// TwinCAT 3 PLC project OC_TwinCAT_EtherCAT
// Title: OC_EtherCAT
// Company: Open Commissioning
// Author: SpiraTec AG
// ProjectVersion: 1.1.8
// Description: Open Commissioning TwinCAT EtherCAT Library
// ProgramVersion: 3.1.4026.19
// libraries:
//   OC_Core, * (Open Commissioning)
//   OC_TwinSAFE, * (Open Commissioning)
//   Tc2_Math, * (Beckhoff Automation GmbH)
//   Tc2_Standard, * (Beckhoff Automation GmbH)
//   Tc2_System, * (Beckhoff Automation GmbH)
//   Tc3_Module, * (Beckhoff Automation GmbH)
//   TcUnit, * (www.tcunit.org)
// project tree:
//   Devices/Drives/DS402/ E_DS402_State.TcDUT, FB_DS402_CSP.TcPOU, FB_DS402_FSM.TcPOU, ST_DS402_CSP_Config.TcDUT, ST_DS402_ControlWord.TcDUT, ST_DS402_CSP_Status.TcDUT, ST_DS402_CSP_Control.TcDUT, ST_DS402_StatusWord.TcDUT
//   Devices/Drives/Mitsubishi/ FB_Mitsubishi_MRJ4TM.TcPOU, ST_Mitsubishi_MRJ4TM_Config.TcDUT, ST_Mitsubishi_MRJ4TM_Control.TcDUT, ST_Mitsubishi_MRJ4TM_Status.TcDUT
//   Devices/Drives/Sercos/ E_Sercos_State.TcDUT, FB_Sercos_FSM.TcPOU, FB_Sercos_VC.TcPOU, ST_Sercos_VC.TcDUT, ST_Sercos_VC_Config.TcDUT, ST_Sercos_VC_Control.TcDUT, ST_Sercos_VC_Status.TcDUT, ST_Sercos_StatusWord.TcDUT, ST_Sercos_ControlWord.TcDUT
//   Devices/Terminals/ FB_Beckhoff_EK1914.TcPOU, FB_Beckhoff_EL5152.TcPOU, FB_Beckhoff_EJ1918.TcPOU, FB_Beckhoff_EL1904.TcPOU, FB_Beckhoff_EL1918.TcPOU, FB_Beckhoff_EL2904.TcPOU, FB_FSOE_19.TcPOU, ST_Baumer_Encoder.TcDUT, ST_Beckhoff_16DI.TcDUT, ST_Beckhoff_16DO.TcDUT (not stored), ST_Beckhoff_2AI.TcDUT (not stored), ST_Beckhoff_4AI.TcDUT (not stored), ST_Beckhoff_4AO.TcDUT, ST_Beckhoff_4DI_4DO.TcDUT (not stored), ST_Beckhoff_8DI.TcDUT, ST_Beckhoff_4DI.TcDUT, ST_Beckhoff_8DI_8DO.TcDUT (not stored), ST_Beckhoff_8DO.TcDUT (not stored), ST_Beckhoff_4DO.TcDUT, ST_Beckhoff_EL3403.TcDUT (not stored), ST_Beckhoff_EL5002.TcDUT (not stored), ST_Beckhoff_EL9110.TcDUT (not stored), ST_Beckhoff_EL9410.TcDUT (not stored), ST_CoE402.TcDUT (not stored), ST_Gefran_GFX4.TcDUT (not stored), ST_Mitsubishi_MRJ4TM.TcDUT, ST_SEW_SimMovitrac.TcDUT (not stored)
//   Devices/Terminals/FB_Beckhoff_EL6001/ E_Beckhoff_EL6001_State.TcDUT, FB_Beckhoff_EL6001.TcPOU
//   / PlcTask.TcTTO
//   Tests/Drives/ FB_Sercos_VC_Test.TcPOU, FB_DS402_FSM_Test.TcPOU, FB_DS402_CSP_Test.TcPOU, FB_Sercos_FSM_Test.TcPOU
//   Tests/Terminals/ FB_Beckhoff_EL5152_Test.TcPOU, FB_Beckhoff_EL6001_Test.TcPOU
//   Tests/ PRG_TEST.TcPOU

CONFIGURATION OC_TwinCAT_EtherCAT
    RESOURCE PLC ON TwinCAT3
        TASK PlcTask(INTERVAL := T#1ms, PRIORITY := 30);
        PROGRAM PRG_TEST WITH PlcTask : PRG_TEST;
    END_RESOURCE
END_CONFIGURATION

// ---- Devices/Drives/DS402/E_DS402_State.TcDUT
{attribute 'qualified_only'}
{attribute 'strict'}
{attribute 'conditionalshow'}
TYPE E_DS402_State :
(
	S0_NotReadyToSwitchOn,
	S1_SwitchOnDisabled,
	S2_ReadyToSwitchOn,
	S3_SwitchedOn,
	S4_OperationEnabled,
	S5_Fault,
	S6_FaultReactionActive,
	S7_QuickStopActive
);
END_TYPE

// ---- Devices/Drives/DS402/ST_DS402_CSP_Config.TcDUT
{attribute 'pack_mode' := '0'}
TYPE ST_DS402_CSP_Config :
STRUCT	
	bForceMode			: BOOL; //Ignore process data from fieldbus.	
	bSwapProcessData	: BOOL; //Reverse process data byte order from/to fieldbus.
	fPositionOffset		: LREAL := 0.0;	
	bSyncOpMode			: BOOL := TRUE;
END_STRUCT
END_TYPE

// ---- Devices/Drives/DS402/ST_DS402_ControlWord.TcDUT
(*
	Object 6040h: Control word (DS402)	
*)
{attribute 'pack_mode' := '0'}
TYPE ST_DS402_ControlWord :
STRUCT
	b0_SwitchOn 					: BIT;
	b1_EnableVoltage				: BIT;
	b2_QuickStop					: BIT;
	b3_EnableOperation				: BIT;
	b4_OperationModeSpecific		: BIT;
	b5_OperationModeSpecific		: BIT;
	b6_OperationModeSpecific		: BIT;
	b7_FaultReset					: BIT;
	b8_Reserved						: BIT;
	b9_Reserved						: BIT;
	b10_Reserved					: BIT;
	b11_Reserved					: BIT;
	b12_Reserved					: BIT;
	b13_Reserved					: BIT;
	b14_Reserved					: BIT;
	b15_Reserved					: BIT;
END_STRUCT
END_TYPE

// ---- Devices/Drives/DS402/ST_DS402_CSP_Status.TcDUT
(*
	Status struct for Cyclic synchronous position mode(CSP)
	0x1A00 (DS402 Statusword)
	0x1A01 (DS402 Position actual value)
	0x1A04 (DS402 Following error actual value)
*)
{attribute 'pack_mode' := '0'}
TYPE ST_DS402_CSP_Status :
STRUCT
	nStatusWord 		: ST_DS402_StatusWord; //0x1A00 (DS402 Statusword)
	nActualPosition		: DINT;	//0x1A01 (DS402 Position actual value) [INC]
	nErrorPosition		: DINT;	//0x1A04 (DS402 Following error actual value) [INC]	
END_STRUCT
END_TYPE

// ---- Devices/Drives/DS402/ST_DS402_CSP_Control.TcDUT
(*
	Control struct for Cyclic synchronous position mode(CSP)
	0x1600 (DS402 Controlword)
	0x1606 (DS402 Target position)
*)
{attribute 'pack_mode' := '0'}
TYPE ST_DS402_CSP_Control :
STRUCT
	nControlWord 		: ST_DS402_ControlWord; //0x1600 (DS402 Controlword)
	nTargetPosition		: DINT;	//DS402 Target position [INC]	
END_STRUCT
END_TYPE

// ---- Devices/Drives/DS402/ST_DS402_StatusWord.TcDUT
(*
	Object 6041h: Status word (DS402)
*)
{attribute 'pack_mode' := '0'}
TYPE ST_DS402_StatusWord :
STRUCT
	b0_ReadyToSwitchOn 				: BIT; 
	b1_SwitchedOn 					: BIT; 
	b2_OperationEnabled 			: BIT; 
	b3_Fault						: BIT; 
	b4_VoltageEnabled				: BIT; 
	b5_QuickStop					: BIT;
	b6_SwitchOnDisabled				: BIT; 
	b7_Warning						: BIT; 
	b8_Synchranisation				: BIT; 
	b9_Remote						: BIT;
	b10_TargetReached				: BIT;
	b11_InternalLimitActive			: BIT; 
	b12_OperationModeSpecific		: BIT; 
	b13_OperationModeSpecific		: BIT; 
	b14_OperationModeSpecific		: BIT; 
	b15_ClosedLoopActive			: BIT;
END_STRUCT
END_TYPE

// ---- Devices/Drives/Mitsubishi/ST_Mitsubishi_MRJ4TM_Config.TcDUT
{attribute 'pack_mode' := '0'}
TYPE ST_Mitsubishi_MRJ4TM_Config :
STRUCT	
	bForceMode			: BOOL; //Ignore process data from fieldbus.	
	bSwapProcessData	: BOOL; //Reverse process data byte order from/to fieldbus.
	fPositionOffset		: LREAL := 0.0;	
	bSyncOpMode			: BOOL := TRUE;
END_STRUCT
END_TYPE

// ---- Devices/Drives/Mitsubishi/ST_Mitsubishi_MRJ4TM_Control.TcDUT
(*
	
*)
{attribute 'pack_mode' := '0'}
TYPE ST_Mitsubishi_MRJ4TM_Control :
STRUCT
	nModesOfOperation 				: SINT;
	nControlWord 					: ST_DS402_ControlWord; //0x1600 (DS402 Controlword)
	nControlID1						: UINT;
	nControlID2						: UINT;
	nControlID3						: UINT;
	nTargetPosit					: DINT;
	nTargetVeloc					: DINT;
	nVelocityLimitValue				: UDINT;
	nTargetTorque					: INT;
	nPositiveTorqueLimitValue		: UINT;
	nNegativeTorqueLimitValue 		: UINT;
	nTouchProbeFunction				: UINT;
END_STRUCT
END_TYPE

// ---- Devices/Drives/Mitsubishi/ST_Mitsubishi_MRJ4TM_Status.TcDUT
(*
	
*)
{attribute 'pack_mode' := '0'}
TYPE ST_Mitsubishi_MRJ4TM_Status :
STRUCT
	nModesOfOperationDisplay 		: SINT;
	nStatusWord 					: ST_DS402_StatusWord; //0x1A00 (DS402 Statusword)
	nStatusDO1						: UINT;
	nStatusDO2						: UINT;
	nStatusDO3						: UINT;
	nPositionActualValue			: DINT;
	nVelocityActualValue			: DINT;
	nFollowingErrorActualValue		: DINT;
	nTorqueActualValue				: INT;
	nTouchProbeStatus				: UINT;
	nTouchProbePos1PosValue			: DINT;
	nTouchProbePos1NegValue			: DINT;
	nTouchProbePos2PosValue			: DINT;
	nTouchProbePos2NegValue			: DINT;
END_STRUCT
END_TYPE

// ---- Devices/Drives/Sercos/E_Sercos_State.TcDUT
{attribute 'qualified_only'}
{attribute 'strict'}
{attribute 'conditionalshow'}
TYPE E_Sercos_State :
(
	S1_NotReadyToSwitchOn,
	S2_SwitchOnDisabled,
	S3_ReadyToSwitchOn,
	S4_SwitchOn,
	S5a_DriveInOperation,
	S5b_Halt,
	S6_QuickStop,
	S7_FaultReactionActive,
	S8_Fault
);
END_TYPE

// ---- Devices/Drives/Sercos/ST_Sercos_VC.TcDUT
{attribute 'pack_mode' := '1'} 
TYPE ST_Sercos_VC :
STRUCT
	stControl		AT %I* : ST_Sercos_VC_Control;
	stStatus		AT %Q* : ST_Sercos_VC_Status;
END_STRUCT
END_TYPE

// ---- Devices/Drives/Sercos/ST_Sercos_VC_Config.TcDUT
{attribute 'pack_mode' := '0'}
TYPE ST_Sercos_VC_Config :
STRUCT	
	bForceMode				: BOOL; //Ignore process data from fieldbus.	
	bSwapProcessData		: BOOL; //Reverse process data byte order from/to fieldbus.	
	bIsLinkOutputVelocity	: BOOL; //If TRUE, link output is velocity value
	fReferenceVelocity 		: REAL := 1000.0;
	fNormalizationFactor	: REAL := 80000;
END_STRUCT
END_TYPE

// ---- Devices/Drives/Sercos/ST_Sercos_VC_Control.TcDUT
(*
	Sercos Velocity Control
	MDT: S-0-0134 Master control word
	MDT: S-0-0036 Velocity command value
*)
{attribute 'pack_mode' := '0'}
TYPE ST_Sercos_VC_Control :
STRUCT
	nControlWord 			: ST_Sercos_ControlWord; //S-0-0134 Master control word
	nVelocityCommand		: DINT;	//S-0-0036 Velocity command value
END_STRUCT
END_TYPE

// ---- Devices/Drives/Sercos/ST_Sercos_VC_Status.TcDUT
(*
	Sercos Velocity Control
	AT: S-0-0135 Drive Status word
	AT: S-0-0051 Position feedback 1 value
*)
{attribute 'pack_mode' := '0'}
TYPE ST_Sercos_VC_Status :
STRUCT
	nStatusWord 			: ST_Sercos_StatusWord; //S-0-0135 Drive Status word
	nPositionFeedback		: DINT;	//S-0-0051 Position feedback 1 value
END_STRUCT
END_TYPE

// ---- Devices/Drives/Sercos/ST_Sercos_StatusWord.TcDUT
(*
	S-0-0135 Drive Status
	https://product-help.schneider-electric.com/Machine%20Expert/V1.2/en/ATV340SUG/ATV340SUG/STI_Software_Setup/STI_Software_Setup-22.htm#XREF_D_SE_0083227_1
*)
{attribute 'pack_mode' := '1'}
TYPE ST_Sercos_StatusWord :
STRUCT
	b0_Reserved 					: BIT;
	b1_Reserved						: BIT;
	b2_Reserved						: BIT;
	b3_CommandProcessing			: BIT; //Status command value processing if 0 = ignored
	b4_Halt							: BIT; //Drive halt, 0 = inactive, 1 = active
	b5_PositionFeedback				: BIT; //Position feedback value status (S-0-0403)
	b6_Reserved						: BIT;
	b7_QuickStop					: BIT; //Quick stop, 0 = inactive, 1 = active
	b8_Reserved						: BIT; //Reserved (=0)
	b9_Reserved						: BIT; //Reserved (=0)
	b10_OperationMode				: BIT; //0 = Primary operation mode
	b11_Reserved					: BIT;
	b12_Warning						: BIT; //Warning, 0 = No warning, 1 = Warning
	b13_Error						: BIT; //Drive shut-down error, 0 = No error, 1 = Error
	b14_ReadyToOperate				: BIT; //00 = Not ready to switch on, 01 = Switch on disabled, main power disabled
	b15_ReadyToOperate				: BIT; //10 = Switch on, 11 = Drive enabled
END_STRUCT
END_TYPE

// ---- Devices/Drives/Sercos/ST_Sercos_ControlWord.TcDUT
(*
	S-0-0134 Drive Control
	https://product-help.schneider-electric.com/Machine%20Expert/V1.2/en/ATV340SUG/ATV340SUG/STI_Software_Setup/STI_Software_Setup-21.htm#XREF_D_SE_0083221_1
*)
{attribute 'pack_mode' := '1'}
TYPE ST_Sercos_ControlWord :
STRUCT
	b0_Reserved 					: BIT;
	b1_Reserved						: BIT;
	b2_Reserved						: BIT;
	b3_Reserved						: BIT;
	b4_Reserved						: BIT;
	b5_Reserved						: BIT;
	b6_Reserved						: BIT;
	b7_Reserved						: BIT;
	b8_Reserved						: BIT; //Reserved (=0)
	b9_Reserved						: BIT; //Reserved (=0)
	b10_OperationMode				: BIT; //0 = Primary operation mode
	b11_Reserved					: BIT;
	b12_Reserved					: BIT; 
	b13_Halt						: BIT; //Drive halt, 1 --> 0 = halt, 0 --> 1 = restart
	b14_Start						: BIT; //Drive start, 1 --> 0 = Stop, 0 -> 1 = Start 
	b15_Enable						: BIT; //Drive enable, 1 --> 0 = drive disabled, 0 -> 1 = drive enabled
END_STRUCT
END_TYPE

// ---- Devices/Terminals/FB_Beckhoff_EL6001/E_Beckhoff_EL6001_State.TcDUT
{attribute 'qualified_only'}
{attribute 'strict'}
TYPE E_Beckhoff_EL6001_State :
(
	INIT,
	READY,
	TRANSMIT, 
	RECEIVE
);
END_TYPE

// ---- Devices/Terminals/ST_Baumer_Encoder.TcDUT
{attribute 'pack_mode' := '1'}
TYPE ST_Baumer_Encoder :
STRUCT
	nPosition		AT %Q*	:	UDINT;
	nWarnings		AT %Q*	:	UINT;
	nSystemTime		AT %Q*	:	UDINT; 
END_STRUCT
END_TYPE

// ---- Devices/Terminals/ST_Beckhoff_16DI.TcDUT
{attribute 'pack_mode' := '1'} 
TYPE ST_Beckhoff_16DI :
STRUCT
	bIn1	AT %Q* : BIT;
	bIn2	AT %Q* : BIT;
	bIn3	AT %Q* : BIT;
	bIn4	AT %Q* : BIT;
	bIn5	AT %Q* : BIT;
	bIn6	AT %Q* : BIT;
	bIn7	AT %Q* : BIT;
	bIn8	AT %Q* : BIT;
	bIn9	AT %Q* : BIT;
	bIn10	AT %Q* : BIT;
	bIn11	AT %Q* : BIT;
	bIn12	AT %Q* : BIT;
	bIn13	AT %Q* : BIT;
	bIn14	AT %Q* : BIT;
	bIn15	AT %Q* : BIT;
	bIn16	AT %Q* : BIT;
END_STRUCT
END_TYPE

// ---- Devices/Terminals/ST_Beckhoff_4AO.TcDUT
{attribute 'pack_mode' := '1'} 
TYPE ST_Beckhoff_4AO :
STRUCT
	nAnalogOut1	AT %I* : UINT;
	nAnalogOut2	AT %I* : UINT;
	nAnalogOut3	AT %I* : UINT;
	nAnalogOut4	AT %I* : UINT;
END_STRUCT
END_TYPE

// ---- Devices/Terminals/ST_Beckhoff_8DI.TcDUT
{attribute 'pack_mode' := '1'} 
TYPE ST_Beckhoff_8DI :
STRUCT
	bIn1	AT %Q* : BIT;
	bIn2	AT %Q* : BIT;
	bIn3	AT %Q* : BIT;
	bIn4	AT %Q* : BIT;
	bIn5	AT %Q* : BIT;
	bIn6	AT %Q* : BIT;
	bIn7	AT %Q* : BIT;
	bIn8	AT %Q* : BIT;
END_STRUCT
END_TYPE

// ---- Devices/Terminals/ST_Beckhoff_4DI.TcDUT
{attribute 'pack_mode' := '1'} 
TYPE ST_Beckhoff_4DI :
STRUCT
	bIn1	AT %Q* : BIT;
	bIn2	AT %Q* : BIT;
	bIn3	AT %Q* : BIT;
	bIn4	AT %Q* : BIT;	
END_STRUCT
END_TYPE

// ---- Devices/Terminals/ST_Beckhoff_4DO.TcDUT
{attribute 'pack_mode' := '1'} 
TYPE ST_Beckhoff_4DO :
STRUCT
	bOut1	AT %I* : BIT;
	bOut2	AT %I* : BIT;
	bOut3	AT %I* : BIT;
	bOut4	AT %I* : BIT;	
END_STRUCT
END_TYPE

// ---- Devices/Terminals/ST_Mitsubishi_MRJ4TM.TcDUT
{attribute 'pack_mode' := '1'} 
TYPE ST_Mitsubishi_MRJ4TM :
STRUCT
	nModesOfOperation 				AT %I* : SINT;
	nControlWord					AT %I* : UINT;
	nControlID1						AT %I* : UINT;
	nControlID2						AT %I* : UINT;
	nControlID3						AT %I* : UINT;
	nTargetPosit					AT %I* : DINT;
	nTargetVeloc					AT %I* : DINT;
	nVelocityLimitValue				AT %I* : UDINT;
	nTargetTorque					AT %I* : INT;
	nPositiveTorqueLimitValue		AT %I* : UINT;
	nNegativeTorqueLimitValue 		AT %I* : UINT;
	nTouchProbeFunction				AT %I* : UINT;
	
	nModesOfOperationDisplay 		AT %Q* : SINT;
	nStatusWord						AT %Q* : UINT;
	nStatusDO1						AT %Q* : UINT;
	nStatusDO2						AT %Q* : UINT;
	nStatusDO3						AT %Q* : UINT;
	nPositionActualValue			AT %Q* : DINT;
	nVelocityActualValue			AT %Q* : DINT;
	nFollowingErrorActualValue		AT %Q* : DINT;
	nTorqueActualValue				AT %Q* : INT;
	nTouchProbeStatus				AT %Q* : UINT;
	nTouchProbePos1PosValue			AT %Q* : DINT;
	nTouchProbePos1NegValue			AT %Q* : DINT;
	nTouchProbePos2PosValue			AT %Q* : DINT;
	nTouchProbePos2NegValue			AT %Q* : DINT;
END_STRUCT
END_TYPE

// ---- Tests/PRG_TEST.TcPOU
PROGRAM PRG_TEST
VAR	
	FB_System	: FB_System;
	FB_Beckhoff_EL5152_Test : FB_Beckhoff_EL5152_Test;
	FB_Beckhoff_EL6001_Test : FB_Beckhoff_EL6001_Test;
	FB_DS402_FSM_Test : FB_DS402_FSM_Test;	
	FB_DS402_CSP_Test : FB_DS402_CSP_Test; 
	FB_Sercos_FSM_Test : FB_Sercos_FSM_Test;
	FB_Sercos_VC_Test : FB_Sercos_VC_Test;
END_VAR

FB_System();
TcUnit.RUN();

END_PROGRAM

// ---- Tests/Terminals/FB_Beckhoff_EL5152_Test.TcPOU
FUNCTION_BLOCK FB_Beckhoff_EL5152_Test EXTENDS TcUnit.FB_TestSuite
VAR
	_fbDevice 	: FB_Beckhoff_EL5152;
	_nExpected 	: UINT;
	_nResult 	: UINT;
END_VAR

TEST('nCounter1');
_nExpected := 111;
_fbDevice.nValue1 := _nExpected;
_fbDevice();
_nResult := _fbDevice.Counter1;
AssertEquals(Expected := _nExpected,
             Actual := _nResult,
             Message := 'nCounter1 value is not correct');	
TEST_FINISHED();

TEST('nCounter2');
_nExpected := 112;
_fbDevice.nValue2 := _nExpected;
_fbDevice();
_nResult := _fbDevice.Counter2;
AssertEquals(Expected := _nExpected,
             Actual := _nResult,
             Message := 'nCounter2 value is not correct');	
TEST_FINISHED();


TEST('nStatus1');
_nExpected := 4;
_fbDevice.Control1 := _nExpected;
_fbDevice();
_nResult := _fbDevice.Status1;
AssertEquals(Expected := _nExpected,
             Actual := _nResult,
             Message := 'nStatus1 value is not correct');	
TEST_FINISHED();

TEST('nStatus2');
_nExpected := 4;
_fbDevice.Control2 := _nExpected;
_fbDevice();
_nResult := _fbDevice.Status2;
AssertEquals(Expected := _nExpected,
             Actual := _nResult,
             Message := 'nStatus2 value is not correct');	
TEST_FINISHED();

END_FUNCTION_BLOCK

// ---- Devices/Terminals/FB_Beckhoff_EL5152.TcPOU
FUNCTION_BLOCK FB_Beckhoff_EL5152
VAR_INPUT
	nValue1		: UINT;
	nValue2		: UINT;
END_VAR
VAR
	nControl1		AT %I* : UINT;
	nSetCounter1	AT %I* : UINT;
	nControl2		AT %I* : UINT;
	nSetCounter2	AT %I* : UINT;
	
	nStatus1		AT %Q* : UINT;
	nCounter1		AT %Q* : UINT;	
	nPeriod1    	AT %Q* : UDINT;
	nStatus2		AT %Q* : UINT;
	nCounter2		AT %Q* : UINT;
	nPeriod2    	AT %Q* : UDINT;
END_VAR

nStatus1.2 := nControl1.2;
nStatus2.2 := nControl2.2;

nCounter1 := nValue1;
nCounter2 := nValue2;

PROPERTY INTERNAL Control1 : UINT
SET
nControl1 := Control1;
END_SET
END_PROPERTY

PROPERTY INTERNAL Control2 : UINT
SET
nControl2 := Control2;
END_SET
END_PROPERTY

PROPERTY INTERNAL Counter1 : UINT
GET
Counter1 := nCounter1;
END_GET
END_PROPERTY

PROPERTY INTERNAL Counter2 : UINT
GET
Counter2 := nCounter2;
END_GET
END_PROPERTY

PROPERTY INTERNAL Period1 : UDINT
GET
Period1 := nPeriod1;
END_GET
END_PROPERTY

PROPERTY INTERNAL Period2 : UDINT
GET
Period2 := nPeriod2;
END_GET
END_PROPERTY

PROPERTY INTERNAL SetCounter1 : UINT
SET
nSetCounter1 := SetCounter1;
END_SET
END_PROPERTY

PROPERTY INTERNAL SetCounter2 : UINT
SET
nSetCounter2 := SetCounter2;
END_SET
END_PROPERTY

PROPERTY INTERNAL Status1 : UINT
GET
Status1 := nStatus1;
END_GET
END_PROPERTY

PROPERTY INTERNAL Status2 : UINT
GET
Status2 := nStatus2;
END_GET
END_PROPERTY

END_FUNCTION_BLOCK

// ---- Tests/Terminals/FB_Beckhoff_EL6001_Test.TcPOU
FUNCTION_BLOCK FB_Beckhoff_EL6001_Test EXTENDS TcUnit.FB_TestSuite
VAR
	_fbDevice 	: FB_Beckhoff_EL6001;
	_nExpected 	: UINT;
	_nResult 	: UINT;
END_VAR

TestProperties();
TestState();

METHOD TestProperties : REFERENCE TO FB_Test
VAR
	bExpected 		: BOOL;
	bResult 		: BOOL;
END_VAR
TEST('TransmitRequest FALSE');
bExpected := FALSE; 
_fbDevice();
_fbDevice.Control := 0;
_fbDevice();
bResult := _fbDevice.TransmitRequest;
AssertEquals(Expected := bExpected,
             Actual := bResult,
             Message := 'TransmitRequest value is not correct');		
TEST_FINISHED();

TEST('TransmitRequest TRUE');
bExpected := TRUE; 
_fbDevice();
_fbDevice.Control := 1;
_fbDevice();
bResult := _fbDevice.TransmitRequest;
AssertEquals(Expected := bExpected,
             Actual := bResult,
             Message := 'TransmitRequest value is not correct');		
TEST_FINISHED();

TEST('ReceiveAccepted FALSE');
bExpected := FALSE; 
_fbDevice();
_fbDevice.Control := 0;
_fbDevice();
bResult := _fbDevice.ReceiveAccepted;
AssertEquals(Expected := bExpected,
             Actual := bResult,
             Message := 'ReceiveAccepted value is not correct');		
TEST_FINISHED();

TEST('ReceiveAccepted TRUE');
bExpected := TRUE; 
_fbDevice();
_fbDevice.Control := 2;
_fbDevice();
bResult := _fbDevice.ReceiveAccepted;
AssertEquals(Expected := bExpected,
             Actual := bResult,
             Message := 'ReceiveAccepted value is not correct');		
TEST_FINISHED();

TEST('InitRequest TRUE');
bExpected := TRUE; 
_fbDevice();
_fbDevice.Control := 4;
_fbDevice();
bResult := _fbDevice.InitRequest;
AssertEquals(Expected := bExpected,
             Actual := bResult,
             Message := 'InitRequest value is not correct');		
TEST_FINISHED();

TEST('SendContinuous TRUE');
bExpected := TRUE; 
_fbDevice.Control := 0;
_fbDevice();
_fbDevice.Control := 9;
_fbDevice();
bResult := _fbDevice.SendContinuous;
AssertEquals(Expected := bExpected,
             Actual := bResult,
             Message := 'SendContinuous value is not correct');		
TEST_FINISHED();
END_METHOD

METHOD TestState : REFERENCE TO FB_Test
VAR
	bResult 		: BOOL;
	nDataSend 		:  ARRAY[0..50] OF BYTE;
END_VAR
TEST('Transition: INIT - READY');
_fbDevice.Control := 0;
_fbDevice.State := E_Beckhoff_EL6001_State.INIT;	
_fbDevice();

AssertTRUE(_fbDevice.State = E_Beckhoff_EL6001_State.READY, 'State value is not correct');
	
TEST_FINISHED();

TEST('Transition: READY - TRANSMIT');
_fbDevice.Control := 0;
_fbDevice.State := E_Beckhoff_EL6001_State.READY;	
_fbDevice();

_fbDevice.Control := 257;
_fbDevice();

AssertTRUE(_fbDevice.State = E_Beckhoff_EL6001_State.TRANSMIT, 'State value is not correct');
	
TEST_FINISHED();

TEST('Transition: READY - RECEIVE');
_fbDevice.Control := 0;
_fbDevice.State := E_Beckhoff_EL6001_State.READY;	
_fbDevice();

_fbDevice.bSend := TRUE;
_fbDevice.pDataIn := ADR(nDataSend);
_fbDevice.nLength := 1;
_fbDevice.Control := 1;
_fbDevice();

_fbDevice.bSend := FALSE;
_fbDevice.nLength := 0;

AssertTRUE(_fbDevice.State = E_Beckhoff_EL6001_State.RECEIVE, 'State value is not correct');
TEST_FINISHED();
END_METHOD

END_FUNCTION_BLOCK

// ---- Devices/Terminals/FB_Beckhoff_EL6001/FB_Beckhoff_EL6001.TcPOU
FUNCTION_BLOCK FB_Beckhoff_EL6001
VAR_INPUT
	bSend				: BOOL;
	nLength				: UINT;
	pDataIn				: POINTER TO BYTE; //Data to send
	pDataOut			: POINTER TO BYTE; //Received data when nDataAvailable > 0.
END_VAR

VAR_OUTPUT
	bBusy				: BOOL;
	nDataAvailable		: INT; //Received bytes. Only available for one cycle.
END_VAR

VAR
	nControl			AT %I* : UINT;
	nDataOut			AT %I* : ARRAY[0..21] OF USINT;
	nStatus				AT %Q* : UINT;
	nDataIn				AT %Q* : ARRAY[0..21] OF USINT;
END_VAR

VAR
	_nControlByte			: BYTE;
	_nOutLength				: BYTE;	
	_bTransmitRequest		: BOOL;
	_bReceiveAccecpted		: BOOL;
	_bInitRequest			: BOOL;
	_bSendContinuous		: BOOL;
	
	_bTransmitAccepted		: BOOL;
	_bReceiveRequest		: BOOL;
	_bInitAccepted			: BOOL;
	_bBufferFull			: BOOL;
	_bParityError			: BOOL;
	_bFramingError			: BOOL;
	_bOverrunError			: BOOL;
	_nInLength				: BYTE;
	
	_nPendingLength			: UINT;
	_nOffsetNext			: UINT;
	
	_eState					: E_Beckhoff_EL6001_State;
	_trigSend				: R_TRIG;
END_VAR

(* Receive control word *)
	_bTransmitRequest 	:= nControl.0 <> _nControlByte.0;
	_bReceiveAccecpted 	:= nControl.1 <> _nControlByte.1;
	_bInitRequest		:= nControl = 4;
	_bSendContinuous		:= nControl.3 AND NOT _nControlByte.0;	
	_nControlByte 		:= F_GetLByte(nControl);
	_nOutLength 			:= F_GetHByte(nControl);

(* Initialize *)
	IF _bInitRequest THEN
		_eState := E_Beckhoff_EL6001_State.INIT;			
	END_IF
	
CASE _eState OF
	E_Beckhoff_EL6001_State.INIT:
		_bTransmitAccepted 	:= FALSE;
		_bReceiveRequest		:= FALSE;
		_bInitAccepted		:= TRUE;
		_bBufferFull			:= FALSE;
		_bParityError		:= FALSE;
		_bFramingError		:= FALSE;
		_bOverrunError		:= FALSE;
		_nInLength			:= 0;
		nDataAvailable		:= 0;
		
		// -> INIT_READY
		IF nControl = 0 THEN
			_bInitAccepted := FALSE;		
			_eState := E_Beckhoff_EL6001_State.READY;
		END_IF

	E_Beckhoff_EL6001_State.READY:
		nDataAvailable := 0;

		// -> TRANSMIT
		IF _bTransmitRequest AND _nOutLength > 0 AND _nOutLength < 23 THEN
			_eState := E_Beckhoff_EL6001_State.TRANSMIT;
			RETURN;
		END_IF
		
		_trigSend(CLK := bSend);
		
		// -> RECEIVE
		IF _trigSend.Q AND nLength > 0 AND pDataIn <> 0 THEN
			_bReceiveRequest := NOT _bReceiveRequest;
			_nPendingLength := nLength;
			_nInLength := UINT_TO_BYTE(MIN(22, _nPendingLength));
			memcpy(ADR(nDataIn), pDataIn, _nInLength);		
			_eState := E_Beckhoff_EL6001_State.RECEIVE;
		END_IF	
		
	E_Beckhoff_EL6001_State.TRANSMIT:
		IF pDataOut <> 0 THEN
			memcpy(pDataOut, ADR(nDataOut), _nOutLength);
		END_IF
		_bTransmitAccepted := NOT _bTransmitAccepted;
		nDataAvailable := _nOutLength;
		_eState := E_Beckhoff_EL6001_State.READY;
		
	E_Beckhoff_EL6001_State.RECEIVE:
		IF _bReceiveAccecpted THEN
			_nOffsetNext := _nInLength;
			_nPendingLength := _nPendingLength - _nOffsetNext;
			IF _nPendingLength = 0 THEN
				_eState := E_Beckhoff_EL6001_State.READY;
			END_IF
			IF _nPendingLength > 0 THEN
				_bReceiveRequest := NOT _bReceiveRequest;
				_nInLength := UINT_TO_BYTE(MIN(22, _nPendingLength));
				memcpy(ADR(nDataIn), pDataIn + _nOffsetNext, _nInLength);
				_eState := E_Beckhoff_EL6001_State.RECEIVE;
			END_IF				
		END_IF
	
END_CASE

bBusy := _eState <> E_Beckhoff_EL6001_State.READY;
	
(* Send status word *)
	nStatus.0			:= _bTransmitAccepted;
	nStatus.1			:= _bReceiveRequest;
	nStatus.2			:= _bInitAccepted;
	nStatus.3			:= _bBufferFull;
	nStatus.4			:= _bParityError;
	nStatus.5			:= _bFramingError;
	nStatus.6			:= _bOverrunError;
	memcpy(ADR(nStatus) + 1, ADR(_nInLength), 1);

PROPERTY INTERNAL BufferFull : BOOl
GET
BufferFull := _bBufferFull;
END_GET
END_PROPERTY

PROPERTY INTERNAL Control : UINT
SET
nControl := Control;
END_SET
END_PROPERTY

PROPERTY INTERNAL FramingError : BOOl
GET
FramingError := _bFramingError;
END_GET
END_PROPERTY

PROPERTY INTERNAL InitAccepted : BOOl
GET
InitAccepted := _bInitAccepted;
END_GET
END_PROPERTY

PROPERTY INTERNAL InitRequest : BOOl
GET
InitRequest := _bInitRequest;
END_GET
END_PROPERTY

PROPERTY INTERNAL OverrunError : BOOl
GET
OverrunError := _bOverrunError;
END_GET
END_PROPERTY

PROPERTY INTERNAL ParityError : BOOl
GET
ParityError := _bParityError;
END_GET
END_PROPERTY

PROPERTY INTERNAL ReceiveAccepted : BOOl
GET
ReceiveAccepted := _bReceiveAccecpted;
END_GET
END_PROPERTY

PROPERTY INTERNAL ReceiveRequest : BOOl
GET
ReceiveRequest := _bReceiveRequest;
END_GET
END_PROPERTY

PROPERTY INTERNAL SendContinuous : BOOl
GET
SendContinuous := _bSendContinuous;
END_GET
END_PROPERTY

PROPERTY INTERNAL State : E_Beckhoff_EL6001_State
GET
State := _eState;
END_GET
SET
_eState := State;
END_SET
END_PROPERTY

PROPERTY INTERNAL TransmitAccepted : BOOl
GET
TransmitAccepted := _bTransmitAccepted;
END_GET
END_PROPERTY

PROPERTY INTERNAL TransmitRequest : BOOl
GET
TransmitRequest := _bTransmitRequest;
END_GET
END_PROPERTY

END_FUNCTION_BLOCK

// ---- Tests/Drives/FB_DS402_FSM_Test.TcPOU
FUNCTION_BLOCK FB_DS402_FSM_Test EXTENDS TcUnit.FB_TestSuite

TestStateS0();
TestStateS1();
TestStateS2();
TestStateS3();
TestStateS4();
TestStateS5();
TestStateS6();
TestStateS7();
TestEnableSequence();

METHOD PRIVATE GetDisableCommand : ST_DS402_ControlWord
GetDisableCommand.b0_SwitchOn := TRUE;
GetDisableCommand.b1_EnableVoltage := TRUE;
GetDisableCommand.b2_QuickStop := TRUE;
GetDisableCommand.b3_EnableOperation := FALSE;
GetDisableCommand.b7_FaultReset := FALSE;
END_METHOD

METHOD PRIVATE GetDisableVoltageCommand : ST_DS402_ControlWord
GetDisableVoltageCommand.b1_EnableVoltage := FALSE;
GetDisableVoltageCommand.b7_FaultReset := FALSE;
END_METHOD

METHOD PRIVATE GetEnableCommand : ST_DS402_ControlWord
GetEnableCommand.b0_SwitchOn := TRUE;
GetEnableCommand.b1_EnableVoltage := TRUE;
GetEnableCommand.b2_QuickStop := TRUE;
GetEnableCommand.b3_EnableOperation := TRUE;
GetEnableCommand.b7_FaultReset := FALSE;
END_METHOD

METHOD PRIVATE GetQuickStopCommand : ST_DS402_ControlWord
GetQuickStopCommand.b2_QuickStop := FALSE;
GetQuickStopCommand.b7_FaultReset := FALSE;
END_METHOD

METHOD PRIVATE GetShotdownCommand : ST_DS402_ControlWord
GetShotdownCommand.b0_SwitchOn := FALSE;
GetShotdownCommand.b1_EnableVoltage := TRUE;
GetShotdownCommand.b2_QuickStop := TRUE;
GetShotdownCommand.b7_FaultReset := FALSE;
END_METHOD

METHOD PRIVATE GetSwitchOnCommand : ST_DS402_ControlWord
GetSwitchOnCommand.b0_SwitchOn := TRUE;
GetSwitchOnCommand.b1_EnableVoltage := TRUE;
GetSwitchOnCommand.b2_QuickStop := TRUE;
GetSwitchOnCommand.b7_FaultReset := FALSE;
END_METHOD

METHOD TestEnableSequence : BOOL
VAR
	fbDS402 			: FB_DS402_FSM;
	stExpectedStatus 	: ST_DS402_StatusWord; 
	nMask 				: WORD;
	nResult 			: WORD;
	bResult 			: BOOL;
	nActualState		: INT;
	nExpectedState		: INT;
END_VAR
TEST('Enable S1');

fbDS402();
nExpectedState := E_DS402_State.S1_SwitchOnDisabled;
nActualState := fbDS402.eState;

AssertEquals(Expected := nExpectedState,
             Actual := nActualState,
             Message := 'State is not correct');	 
TEST_FINISHED();

TEST('Enable S2');
fbDS402.stControl.b1_EnableVoltage := TRUE;
fbDS402.stControl.b2_QuickStop := TRUE;

fbDS402();
nExpectedState := E_DS402_State.S2_ReadyToSwitchOn;
nActualState := fbDS402.eState;

AssertEquals(Expected := nExpectedState,
             Actual := nActualState,
             Message := 'State is not correct');	 
TEST_FINISHED();

TEST('Enable S3');
fbDS402.stControl.b0_SwitchOn := TRUE;

fbDS402();
nExpectedState := E_DS402_State.S3_SwitchedOn;
nActualState := fbDS402.eState;

AssertEquals(Expected := nExpectedState,
             Actual := nActualState,
             Message := 'State is not correct');	 
TEST_FINISHED();

TEST('Enable S4');
fbDS402.stControl.b3_EnableOperation := TRUE;

fbDS402();
nExpectedState := E_DS402_State.S4_OperationEnabled;
nActualState := fbDS402.eState;

AssertEquals(Expected := nExpectedState,
             Actual := nActualState,
             Message := 'State is not correct');	 
TEST_FINISHED();

TEST('Disable S4');
fbDS402.stControl.b3_EnableOperation := FALSE;

fbDS402();
nExpectedState := E_DS402_State.S3_SwitchedOn;
nActualState := fbDS402.eState;

AssertEquals(Expected := nExpectedState,
             Actual := nActualState,
             Message := 'State is not correct');	 
TEST_FINISHED();

TEST('Disable S3');
fbDS402.stControl.b0_SwitchOn := FALSE;

fbDS402();
nExpectedState := E_DS402_State.S2_ReadyToSwitchOn;
nActualState := fbDS402.eState;

AssertEquals(Expected := nExpectedState,
             Actual := nActualState,
             Message := 'State is not correct');	 
TEST_FINISHED();

TEST('Disable S2');
fbDS402.stControl.b1_EnableVoltage := FALSE;
fbDS402.stControl.b2_QuickStop := FALSE;

fbDS402();
nExpectedState := E_DS402_State.S1_SwitchOnDisabled;
nActualState := fbDS402.eState;

AssertEquals(Expected := nExpectedState,
             Actual := nActualState,
             Message := 'State is not correct');	 
TEST_FINISHED();
END_METHOD

METHOD TestStateS0 : BOOL
VAR
	fbDS402 			: FB_DS402_FSM;
	stExpectedStatus 	: ST_DS402_StatusWord; 
	nMask 				: WORD;
	nResult 			: WORD;
	bResult 			: BOOL;
	nActualState		: INT;
	nExpectedState		: INT;
END_VAR
TEST('Set State S0');
fbDS402.eState := E_DS402_State.S0_NotReadyToSwitchOn;
fbDS402();

stExpectedStatus.b0_ReadyToSwitchOn 		:= FALSE;
stExpectedStatus.b1_SwitchedOn 				:= FALSE;
stExpectedStatus.b2_OperationEnabled		:= FALSE;
stExpectedStatus.b3_Fault					:= FALSE;
stExpectedStatus.b4_VoltageEnabled			:= FALSE;
stExpectedStatus.b6_SwitchOnDisabled 		:= FALSE;

MEMCPY(ADR(nMask), ADR(stExpectedStatus), 2);
nResult := (2#01011111 AND fbDS402.nStatus);

AssertEquals(Expected := nMask,
             Actual := nResult,
             Message := 'Value is not correct');	 
TEST_FINISHED();

TEST('Transition S0>S1');
fbDS402.eState := E_DS402_State.S0_NotReadyToSwitchOn;
fbDS402();
fbDS402();

nExpectedState := E_DS402_State.S1_SwitchOnDisabled;
nActualState := fbDS402.eState;

AssertEquals(Expected := nExpectedState,
             Actual := nActualState,
             Message := 'State is not correct');	 
TEST_FINISHED();
END_METHOD

METHOD TestStateS1 : BOOL
VAR
	fbDS402 			: FB_DS402_FSM;
	stExpectedStatus 	: ST_DS402_StatusWord; 
	nMask 				: WORD;
	nResult 			: WORD;
	bResult 			: BOOL;
	nActualState		: INT;
	nExpectedState		: INT;
END_VAR
TEST('Set State S1');
fbDS402.eState := E_DS402_State.S1_SwitchOnDisabled;
fbDS402();

stExpectedStatus.b0_ReadyToSwitchOn 		:= FALSE;
stExpectedStatus.b1_SwitchedOn 				:= FALSE;
stExpectedStatus.b2_OperationEnabled		:= FALSE;
stExpectedStatus.b3_Fault					:= FALSE;
stExpectedStatus.b4_VoltageEnabled			:= FALSE;
stExpectedStatus.b6_SwitchOnDisabled 		:= TRUE;

MEMCPY(ADR(nMask), ADR(stExpectedStatus), 2);
nResult := (2#01011111 AND fbDS402.nStatus);

AssertEquals(Expected := nMask,
             Actual := nResult,
             Message := 'Value is not correct');	 
TEST_FINISHED();

TEST('Transition S1>S2');
fbDS402.eState := E_DS402_State.S1_SwitchOnDisabled;
fbDS402.stControl := GetShotdownCommand();
fbDS402();

nExpectedState := E_DS402_State.S2_ReadyToSwitchOn;
nActualState := fbDS402.eState;


AssertEquals(Expected := nExpectedState,
             Actual := nActualState,
             Message := 'State is not correct');	 
TEST_FINISHED();
END_METHOD

METHOD TestStateS2 : BOOL
VAR
	fbDS402 			: FB_DS402_FSM;
	stExpectedStatus 	: ST_DS402_StatusWord; 
	nMask 				: WORD;
	nResult 			: WORD;
	bResult 			: BOOL;
	nActualState		: INT;
	nExpectedState		: INT;
END_VAR
TEST('Set State S2');
fbDS402.eState := E_DS402_State.S2_ReadyToSwitchOn;
fbDS402();

stExpectedStatus.b0_ReadyToSwitchOn 		:= TRUE;
stExpectedStatus.b1_SwitchedOn 				:= FALSE;
stExpectedStatus.b2_OperationEnabled		:= FALSE;
stExpectedStatus.b3_Fault					:= FALSE;
stExpectedStatus.b4_VoltageEnabled			:= TRUE;
stExpectedStatus.b5_QuickStop 				:= TRUE; 
stExpectedStatus.b6_SwitchOnDisabled 		:= FALSE;

MEMCPY(ADR(nMask), ADR(stExpectedStatus), 2);
nResult := (2#01111111 AND fbDS402.nStatus);

AssertEquals(Expected := nMask,
             Actual := nResult,
             Message := 'Value is not correct');	 
TEST_FINISHED();

TEST('Transition S2>S6');
fbDS402.eState := E_DS402_State.S2_ReadyToSwitchOn;
fbDS402.bError := TRUE;
fbDS402();
fbDS402.ResetError();

nExpectedState := E_DS402_State.S6_FaultReactionActive;
nActualState := fbDS402.eState;

AssertEquals(Expected := nExpectedState,
             Actual := nActualState,
             Message := 'State is not correct');	 
TEST_FINISHED();

TEST('Transition S2>S1_1');
fbDS402.eState := E_DS402_State.S2_ReadyToSwitchOn;
fbDS402.stControl := GetDisableVoltageCommand();
fbDS402();

nExpectedState := E_DS402_State.S1_SwitchOnDisabled;
nActualState := fbDS402.eState;

AssertEquals(Expected := nExpectedState,
             Actual := nActualState,
             Message := 'State is not correct');	 
TEST_FINISHED();

TEST('Transition S2>S1_2');
fbDS402.eState := E_DS402_State.S2_ReadyToSwitchOn;
fbDS402.stControl := GetQuickStopCommand();
fbDS402.stControl.b1_EnableVoltage := TRUE;
fbDS402();

nExpectedState := E_DS402_State.S1_SwitchOnDisabled;
nActualState := fbDS402.eState;

AssertEquals(Expected := nExpectedState,
             Actual := nActualState,
             Message := 'State is not correct');	 
TEST_FINISHED();

TEST('Transition S2>S3');
fbDS402.eState := E_DS402_State.S2_ReadyToSwitchOn;
fbDS402.stControl := GetSwitchOnCommand();
fbDS402();

nExpectedState := E_DS402_State.S3_SwitchedOn;
nActualState := fbDS402.eState;

AssertEquals(Expected := nExpectedState,
             Actual := nActualState,
             Message := 'State is not correct');	 
TEST_FINISHED();
END_METHOD

METHOD TestStateS3 : BOOL
VAR
	fbDS402 			: FB_DS402_FSM;
	stExpectedStatus 	: ST_DS402_StatusWord; 
	nMask 				: WORD;
	nResult 			: WORD;
	bResult 			: BOOL;
	nActualState		: INT;
	nExpectedState		: INT;
END_VAR
TEST('Set State S3');
fbDS402.eState := E_DS402_State.S3_SwitchedOn;
fbDS402();

stExpectedStatus.b0_ReadyToSwitchOn 		:= TRUE;
stExpectedStatus.b1_SwitchedOn 				:= TRUE;
stExpectedStatus.b2_OperationEnabled		:= FALSE;
stExpectedStatus.b3_Fault					:= FALSE;
stExpectedStatus.b5_QuickStop 				:= TRUE; 
stExpectedStatus.b6_SwitchOnDisabled 		:= FALSE;

MEMCPY(ADR(nMask), ADR(stExpectedStatus), 2);
nResult := (2#01101111 AND fbDS402.nStatus);

AssertEquals(Expected := nMask,
             Actual := nResult,
             Message := 'Value is not correct');	 
TEST_FINISHED();

TEST('Transition S3>S6');
fbDS402.eState := E_DS402_State.S3_SwitchedOn;
fbDS402.bError := TRUE;
fbDS402();
fbDS402.ResetError();

nExpectedState := E_DS402_State.S6_FaultReactionActive;
nActualState := fbDS402.eState;

AssertEquals(Expected := nExpectedState,
             Actual := nActualState,
             Message := 'State is not correct');	 
TEST_FINISHED();

TEST('Transition S3>S1_1');
fbDS402.eState := E_DS402_State.S3_SwitchedOn;
fbDS402.stControl := GetDisableVoltageCommand();
fbDS402();

nExpectedState := E_DS402_State.S1_SwitchOnDisabled;
nActualState := fbDS402.eState;

AssertEquals(Expected := nExpectedState,
             Actual := nActualState,
             Message := 'State is not correct');	 
TEST_FINISHED();

TEST('Transition S3>S1_2');
fbDS402.eState := E_DS402_State.S3_SwitchedOn;
fbDS402.stControl := GetQuickStopCommand();
fbDS402.stControl.b1_EnableVoltage := TRUE;
fbDS402();

nExpectedState := E_DS402_State.S1_SwitchOnDisabled;
nActualState := fbDS402.eState;

AssertEquals(Expected := nExpectedState,
             Actual := nActualState,
             Message := 'State is not correct');	 
TEST_FINISHED();

TEST('Transition S3>S2');
fbDS402.eState := E_DS402_State.S3_SwitchedOn;
fbDS402.stControl := GetShotdownCommand();
fbDS402();

nExpectedState := E_DS402_State.S2_ReadyToSwitchOn;
nActualState := fbDS402.eState;

AssertEquals(Expected := nExpectedState,
             Actual := nActualState,
             Message := 'State is not correct');	 
TEST_FINISHED();

TEST('Transition S3>S4');
fbDS402.eState := E_DS402_State.S3_SwitchedOn;
fbDS402.stControl := GetEnableCommand();
fbDS402();

nExpectedState := E_DS402_State.S4_OperationEnabled;
nActualState := fbDS402.eState;

AssertEquals(Expected := nExpectedState,
             Actual := nActualState,
             Message := 'State is not correct');	 
TEST_FINISHED();
END_METHOD

METHOD TestStateS4 : BOOL
VAR
	fbDS402 			: FB_DS402_FSM;
	stExpectedStatus 	: ST_DS402_StatusWord; 
	nMask 				: WORD;
	nResult 			: WORD;
	bResult 			: BOOL;
	nActualState		: INT;
	nExpectedState		: INT;
END_VAR
TEST('Set State S4');
fbDS402.eState := E_DS402_State.S4_OperationEnabled;
fbDS402();

stExpectedStatus.b0_ReadyToSwitchOn 		:= TRUE;
stExpectedStatus.b1_SwitchedOn 				:= TRUE;
stExpectedStatus.b2_OperationEnabled		:= TRUE;
stExpectedStatus.b3_Fault					:= FALSE;
stExpectedStatus.b5_QuickStop 				:= TRUE; 
stExpectedStatus.b6_SwitchOnDisabled 		:= FALSE;

MEMCPY(ADR(nMask), ADR(stExpectedStatus), 2);
nResult := (2#01101111 AND fbDS402.nStatus);

AssertEquals(Expected := nMask,
             Actual := nResult,
             Message := 'Value is not correct');	 
TEST_FINISHED();

TEST('Transition S4>S6');
fbDS402.eState := E_DS402_State.S4_OperationEnabled;
fbDS402.bError := TRUE;
fbDS402();
fbDS402.ResetError();

nExpectedState := E_DS402_State.S6_FaultReactionActive;
nActualState := fbDS402.eState;

AssertEquals(Expected := nExpectedState,
             Actual := nActualState,
             Message := 'State is not correct');	 
TEST_FINISHED();

TEST('Transition S4>S1');
fbDS402.eState := E_DS402_State.S4_OperationEnabled;
fbDS402.stControl := GetDisableVoltageCommand();
fbDS402();

nExpectedState := E_DS402_State.S1_SwitchOnDisabled;
nActualState := fbDS402.eState;

AssertEquals(Expected := nExpectedState,
             Actual := nActualState,
             Message := 'State is not correct');	 
TEST_FINISHED();

TEST('Transition S4>S2');
fbDS402.eState := E_DS402_State.S4_OperationEnabled;
fbDS402.stControl := GetShotdownCommand();
fbDS402();

nExpectedState := E_DS402_State.S2_ReadyToSwitchOn;
nActualState := fbDS402.eState;

AssertEquals(Expected := nExpectedState,
             Actual := nActualState,
             Message := 'State is not correct');	 
TEST_FINISHED();

TEST('Transition S4>S3');
fbDS402.eState := E_DS402_State.S4_OperationEnabled;
fbDS402.stControl := GetDisableCommand();
fbDS402();

nExpectedState := E_DS402_State.S3_SwitchedOn;
nActualState := fbDS402.eState;

AssertEquals(Expected := nExpectedState,
             Actual := nActualState,
             Message := 'State is not correct');	 
TEST_FINISHED();

TEST('Transition S4>S7');
fbDS402.eState := E_DS402_State.S4_OperationEnabled;
fbDS402.stControl := GetQuickStopCommand();
fbDS402.stControl.b1_EnableVoltage := TRUE;
fbDS402();

nExpectedState := E_DS402_State.S7_QuickStopActive;
nActualState := fbDS402.eState;

AssertEquals(Expected := nExpectedState,
             Actual := nActualState,
             Message := 'State is not correct');	 
TEST_FINISHED();
END_METHOD

METHOD TestStateS5 : BOOL
VAR
	fbDS402 			: FB_DS402_FSM;
	stExpectedStatus 	: ST_DS402_StatusWord; 
	nMask 				: WORD;
	nResult 			: WORD;
	bResult 			: BOOL;
	nActualState		: INT;
	nExpectedState		: INT;
END_VAR
TEST('Set State S5');
fbDS402.eState := E_DS402_State.S5_Fault;
fbDS402();

stExpectedStatus.b0_ReadyToSwitchOn 		:= FALSE;
stExpectedStatus.b1_SwitchedOn 				:= FALSE;
stExpectedStatus.b2_OperationEnabled		:= FALSE;
stExpectedStatus.b3_Fault					:= TRUE;
stExpectedStatus.b6_SwitchOnDisabled 		:= FALSE;

MEMCPY(ADR(nMask), ADR(stExpectedStatus), 2);
nResult := (2#01001111 AND fbDS402.nStatus);

AssertEquals(Expected := nMask,
             Actual := nResult,
             Message := 'Value is not correct');	 
TEST_FINISHED();

TEST('Transition S5>S1');
fbDS402.eState := E_DS402_State.S5_Fault;
fbDS402.stControl.b7_FaultReset := TRUE;
fbDS402();
fbDS402.stControl.b7_FaultReset := FALSE;

nExpectedState := E_DS402_State.S1_SwitchOnDisabled;
nActualState := fbDS402.eState;

AssertEquals(Expected := nExpectedState,
             Actual := nActualState,
             Message := 'State is not correct');	 
TEST_FINISHED();
END_METHOD

METHOD TestStateS6 : BOOL
VAR
	fbDS402 			: FB_DS402_FSM;
	stExpectedStatus 	: ST_DS402_StatusWord; 
	nMask 				: WORD;
	nResult 			: WORD;
	bResult 			: BOOL;
	nActualState		: INT;
	nExpectedState		: INT;
END_VAR
TEST('Set State S6');
fbDS402.eState := E_DS402_State.S6_FaultReactionActive;
fbDS402();

stExpectedStatus.b0_ReadyToSwitchOn 		:= TRUE;
stExpectedStatus.b1_SwitchedOn 				:= TRUE;
stExpectedStatus.b2_OperationEnabled		:= TRUE;
stExpectedStatus.b3_Fault					:= TRUE;
stExpectedStatus.b6_SwitchOnDisabled 		:= FALSE;

MEMCPY(ADR(nMask), ADR(stExpectedStatus), 2);
nResult := (2#01001111 AND fbDS402.nStatus);

AssertEquals(Expected := nMask,
             Actual := nResult,
             Message := 'Value is not correct');	 
TEST_FINISHED();

TEST('Transition S6>S5');
fbDS402.eState := E_DS402_State.S6_FaultReactionActive;
fbDS402();

nExpectedState := E_DS402_State.S5_Fault;
nActualState := fbDS402.eState;

AssertEquals(Expected := nExpectedState,
             Actual := nActualState,
             Message := 'State is not correct');	 
TEST_FINISHED();
END_METHOD

METHOD TestStateS7 : BOOL
VAR
	fbDS402 			: FB_DS402_FSM;
	stExpectedStatus 	: ST_DS402_StatusWord; 
	nMask 				: WORD;
	nResult 			: WORD;
	bResult 			: BOOL;
	nActualState		: INT;
	nExpectedState		: INT;
END_VAR
TEST('Set State S7');
fbDS402.eState := E_DS402_State.S7_QuickStopActive;
fbDS402();

stExpectedStatus.b0_ReadyToSwitchOn 		:= TRUE;
stExpectedStatus.b1_SwitchedOn 				:= TRUE;
stExpectedStatus.b2_OperationEnabled		:= TRUE;
stExpectedStatus.b3_Fault					:= FALSE;
stExpectedStatus.b5_QuickStop				:= FALSE;
stExpectedStatus.b6_SwitchOnDisabled 		:= FALSE;

MEMCPY(ADR(nMask), ADR(stExpectedStatus), 2);
nResult := (2#01101111 AND fbDS402.nStatus);

AssertEquals(Expected := nMask,
             Actual := nResult,
             Message := 'Value is not correct');	 
TEST_FINISHED();

TEST('Transition S7>S1');
fbDS402.eState := E_DS402_State.S7_QuickStopActive;
fbDS402.stControl := GetDisableVoltageCommand();
fbDS402();

nExpectedState := E_DS402_State.S1_SwitchOnDisabled;
nActualState := fbDS402.eState;

AssertEquals(Expected := nExpectedState,
             Actual := nActualState,
             Message := 'State is not correct');	 
TEST_FINISHED();

TEST('Transition S7>S4');
fbDS402.eState := E_DS402_State.S7_QuickStopActive;
fbDS402.stControl := GetEnableCommand();
fbDS402();

nExpectedState := E_DS402_State.S4_OperationEnabled;
nActualState := fbDS402.eState;

AssertEquals(Expected := nExpectedState,
             Actual := nActualState,
             Message := 'State is not correct');	 
TEST_FINISHED();
END_METHOD

END_FUNCTION_BLOCK

// ---- Devices/Drives/DS402/FB_DS402_FSM.TcPOU
(*
	DS402 Finite State Machine General
*)
FUNCTION_BLOCK FB_DS402_FSM
VAR_INPUT	
	stControl					: ST_DS402_ControlWord;
END_VAR

VAR_OUTPUT	
	stStatus					: ST_DS402_StatusWord;	
END_VAR

VAR	
	_eState 					: E_DS402_State := E_DS402_State.S0_NotReadyToSwitchOn;	
	_rTrig_QuickStop 			: R_TRIG;
	_rTrig_Reset 				: R_TRIG;
	_bError						: BOOL;
END_VAR

_rTrig_QuickStop(CLK := stControl.b2_QuickStop);
_rTrig_Reset(CLK := stControl.b7_FaultReset);

CASE _eState OF
	E_DS402_State.S0_NotReadyToSwitchOn : S0_NotReadyToSwitchOn();
	E_DS402_State.S1_SwitchOnDisabled : S1_SwitchOnDisabled();
	E_DS402_State.S2_ReadyToSwitchOn : S2_ReadyToSwitchOn();
	E_DS402_State.S3_SwitchedOn : S3_SwitchedOn();
	E_DS402_State.S4_OperationEnabled : S4_OperationEnabled();
	E_DS402_State.S5_Fault : S5_Fault();	
	E_DS402_State.S6_FaultReactionActive : S6_FaultReactionActive();	
	E_DS402_State.S7_QuickStopActive : S7_QuickStopActive();			
END_CASE

PROPERTY PUBLIC bError : BOOL
GET
bError := _bError;
END_GET
SET
IF bError AND NOT _bError THEN
	_bError := TRUE;
END_IF
END_SET
END_PROPERTY

PROPERTY eState : E_DS402_State
GET
eState := _eState;
END_GET
SET
_eState := eState;
END_SET
END_PROPERTY

METHOD PRIVATE IsDisableOperation : BOOL
IsDisableOperation := 
stControl.b0_SwitchOn 
AND stControl.b1_EnableVoltage 
AND stControl.b2_QuickStop 
AND NOT stControl.b3_EnableOperation
AND NOT stControl.b7_FaultReset;
END_METHOD

METHOD PRIVATE IsDisableVoltage : BOOL
IsDisableVoltage := 
NOT stControl.b1_EnableVoltage
AND NOT stControl.b7_FaultReset;
END_METHOD

METHOD PRIVATE IsEnableOperation : BOOL
IsEnableOperation := 
stControl.b0_SwitchOn 
AND stControl.b1_EnableVoltage 
AND stControl.b2_QuickStop 
AND stControl.b3_EnableOperation
AND NOT stControl.b7_FaultReset;
END_METHOD

METHOD PRIVATE IsFaultReset : BOOL
IsFaultReset := _rTrig_Reset.Q;
END_METHOD

METHOD PRIVATE IsQuickStop : BOOL
IsQuickStop := 
NOT stControl.b2_QuickStop
AND NOT stControl.b7_FaultReset;
END_METHOD

METHOD PRIVATE IsShutdown : BOOL
IsShutdown := 
NOT stControl.b0_SwitchOn 
AND stControl.b1_EnableVoltage 
AND stControl.b2_QuickStop
AND NOT stControl.b7_FaultReset;
END_METHOD

METHOD PRIVATE IsSwitchOn : BOOL
IsSwitchOn := 
stControl.b0_SwitchOn 
AND stControl.b1_EnableVoltage 
AND stControl.b2_QuickStop
AND NOT stControl.b7_FaultReset;
END_METHOD

PROPERTY nControl : WORD
GET
nControl.0	:= stControl.b0_SwitchOn;					         
nControl.1	:= stControl.b1_EnableVoltage;				      	
nControl.2	:= stControl.b2_QuickStop;					         	
nControl.3	:= stControl.b3_EnableOperation;			     	
nControl.4	:= stControl.b4_OperationModeSpecific;			
nControl.5	:= stControl.b5_OperationModeSpecific;			
nControl.6	:= stControl.b6_OperationModeSpecific;			
nControl.7	:= stControl.b7_FaultReset;					        	
nControl.8	:= stControl.b8_Reserved;					          	
nControl.9	:= stControl.b9_Reserved;					          
nControl.10	:= stControl.b10_Reserved;					         	
nControl.11	:= stControl.b11_Reserved;					         	
nControl.12	:= stControl.b12_Reserved;					         	
nControl.13	:= stControl.b13_Reserved;					         	
nControl.14	:= stControl.b14_Reserved;					         	
nControl.15 := stControl.b15_Reserved;
END_GET
SET
stControl.b0_SwitchOn 					:= 	nControl.0;	
stControl.b1_EnableVoltage				:= 	nControl.1;		
stControl.b2_QuickStop					:= 	nControl.2;		
stControl.b3_EnableOperation			:= 	nControl.3;		
stControl.b4_OperationModeSpecific		:= 	nControl.4;		
stControl.b5_OperationModeSpecific		:= 	nControl.5;		
stControl.b6_OperationModeSpecific		:= 	nControl.6;		
stControl.b7_FaultReset					:= 	nControl.7;		
stControl.b8_Reserved					:= 	nControl.8;		
stControl.b9_Reserved					:= 	nControl.9;		
stControl.b10_Reserved					:= 	nControl.10;		
stControl.b11_Reserved					:= 	nControl.11;		
stControl.b12_Reserved					:= 	nControl.12;		
stControl.b13_Reserved					:= 	nControl.13;		
stControl.b14_Reserved					:= 	nControl.14;		
stControl.b15_Reserved					:= 	nControl.15;
END_SET
END_PROPERTY

PROPERTY nStatus : WORD
GET
nStatus.0 := stStatus.b0_ReadyToSwitchOn; 			
nStatus.1 := stStatus.b1_SwitchedOn; 				
nStatus.2 := stStatus.b2_OperationEnabled;			
nStatus.3 := stStatus.b3_Fault;					
nStatus.4 := stStatus.b4_VoltageEnabled;
nStatus.5 := stStatus.b5_QuickStop;
nStatus.6 := stStatus.b6_SwitchOnDisabled;			
nStatus.7 := stStatus.b7_Warning;					
nStatus.8 := stStatus.b8_Synchranisation;			
nStatus.9 := stStatus.b9_Remote;			
nStatus.10 := stStatus.b10_TargetReached;				
nStatus.11 := stStatus.b11_InternalLimitActive;		
nStatus.12 := stStatus.b12_OperationModeSpecific;			
nStatus.13 := stStatus.b13_OperationModeSpecific;			
nStatus.14 := stStatus.b14_OperationModeSpecific;			
nStatus.15 := stStatus.b15_ClosedLoopActive;
END_GET
END_PROPERTY

METHOD INTERNAL ResetError : BOOL
_bError := FALSE;
END_METHOD

METHOD PRIVATE S0_NotReadyToSwitchOn : BOOL
VAR_INPUT
END_VAR
stStatus.b0_ReadyToSwitchOn 		:= FALSE;
stStatus.b1_SwitchedOn 				:= FALSE;
stStatus.b2_OperationEnabled		:= FALSE;
stStatus.b3_Fault					:= FALSE;
stStatus.b4_VoltageEnabled			:= FALSE;
stStatus.b6_SwitchOnDisabled 		:= FALSE;

_eState := E_DS402_State.S1_SwitchOnDisabled;
END_METHOD

METHOD PRIVATE S1_SwitchOnDisabled : BOOL
VAR_INPUT
END_VAR
stStatus.b0_ReadyToSwitchOn 		:= FALSE;
stStatus.b1_SwitchedOn				:= FALSE;
stStatus.b2_OperationEnabled 		:= FALSE;
stStatus.b3_Fault 					:= FALSE;
stStatus.b4_VoltageEnabled			:= FALSE;
stStatus.b6_SwitchOnDisabled 		:= TRUE;

IF IsShutdown() THEN
	_eState := E_DS402_State.S2_ReadyToSwitchOn;
END_IF
END_METHOD

METHOD PRIVATE S2_ReadyToSwitchOn : BOOL
VAR_INPUT
END_VAR
stStatus.b0_ReadyToSwitchOn 		:= TRUE;
stStatus.b1_SwitchedOn 				:= FALSE;
stStatus.b2_OperationEnabled 		:= FALSE;
stStatus.b3_Fault 					:= FALSE;
stStatus.b4_VoltageEnabled			:= TRUE;
stStatus.b5_QuickStop 				:= TRUE; 
stStatus.b6_SwitchOnDisabled 		:= FALSE;

IF _bError THEN
	_eState := E_DS402_State.S6_FaultReactionActive;
	RETURN;
END_IF

IF IsDisableVoltage() OR IsQuickStop() THEN
	_eState := E_DS402_State.S1_SwitchOnDisabled;
	RETURN;
END_IF

IF IsSwitchOn() THEN
	_eState := E_DS402_State.S3_SwitchedOn;
	RETURN;
END_IF
END_METHOD

METHOD PRIVATE S3_SwitchedOn : BOOL
VAR_INPUT
END_VAR
stStatus.b0_ReadyToSwitchOn 		:= TRUE;
stStatus.b1_SwitchedOn 				:= TRUE;
stStatus.b2_OperationEnabled 		:= FALSE;
stStatus.b3_Fault 					:= FALSE;
stStatus.b5_QuickStop 				:= TRUE; 
stStatus.b6_SwitchOnDisabled 		:= FALSE;

IF _bError THEN
	_eState := E_DS402_State.S6_FaultReactionActive;
	RETURN;
END_IF

IF IsDisableVoltage() OR IsQuickStop() THEN
	_eState := E_DS402_State.S1_SwitchOnDisabled;
	RETURN;
END_IF

IF IsShutdown() THEN
	_eState := E_DS402_State.S2_ReadyToSwitchOn;
	RETURN;
END_IF

IF IsEnableOperation() THEN
	_eState := E_DS402_State.S4_OperationEnabled;
	RETURN;
END_IF
END_METHOD

METHOD PRIVATE S4_OperationEnabled : BOOL
VAR_INPUT
END_VAR
stStatus.b0_ReadyToSwitchOn				:= TRUE;
stStatus.b1_SwitchedOn 					:= TRUE;
stStatus.b2_OperationEnabled 			:= TRUE;
stStatus.b3_Fault 						:= FALSE;
stStatus.b5_QuickStop 					:= TRUE; 
stStatus.b6_SwitchOnDisabled 			:= FALSE;

IF _bError THEN
	_eState := E_DS402_State.S6_FaultReactionActive;
	RETURN;
END_IF

IF IsDisableVoltage() THEN
	_eState := E_DS402_State.S1_SwitchOnDisabled;
	RETURN;
END_IF

IF IsShutdown() THEN
	_eState := E_DS402_State.S2_ReadyToSwitchOn;
	RETURN;
END_IF

IF IsQuickStop() THEN
	_eState := E_DS402_State.S7_QuickStopActive;
	RETURN;
END_IF

IF IsDisableOperation() THEN
	_eState := E_DS402_State.S3_SwitchedOn;
	RETURN;
END_IF
END_METHOD

METHOD PRIVATE S5_Fault : BOOL
VAR_INPUT
END_VAR
stStatus.b0_ReadyToSwitchOn 		:= FALSE;
stStatus.b1_SwitchedOn				:= FALSE;
stStatus.b2_OperationEnabled 		:= FALSE;
stStatus.b3_Fault 					:= TRUE;
stStatus.b6_SwitchOnDisabled 		:= FALSE;

IF IsFaultReset() THEN
	_bError := FALSE;
	_eState := E_DS402_State.S1_SwitchOnDisabled;
	RETURN;
END_IF
END_METHOD

METHOD PRIVATE S6_FaultReactionActive : BOOL
VAR_INPUT
END_VAR
stStatus.b0_ReadyToSwitchOn 		:= TRUE;
stStatus.b1_SwitchedOn 				:= TRUE;
stStatus.b2_OperationEnabled 		:= TRUE;
stStatus.b3_Fault 					:= TRUE;
stStatus.b6_SwitchOnDisabled 		:= FALSE;

_eState := E_DS402_State.S5_Fault;
END_METHOD

METHOD PRIVATE S7_QuickStopActive : BOOL
VAR_INPUT
END_VAR
stStatus.b0_ReadyToSwitchOn 		:= TRUE;
stStatus.b1_SwitchedOn 				:= TRUE;
stStatus.b2_OperationEnabled 		:= TRUE;
stStatus.b3_Fault 					:= FALSE;
stStatus.b5_QuickStop 				:= FALSE; 
stStatus.b6_SwitchOnDisabled		:= FALSE;

IF IsDisableVoltage() THEN
	_eState := E_DS402_State.S1_SwitchOnDisabled;
	RETURN;
END_IF

IF IsEnableOperation() THEN
	_eState := E_DS402_State.S4_OperationEnabled;
	RETURN;
END_IF
END_METHOD

END_FUNCTION_BLOCK

// ---- Tests/Drives/FB_DS402_CSP_Test.TcPOU
FUNCTION_BLOCK FB_DS402_CSP_Test EXTENDS TcUnit.FB_TestSuite

TestEnable();
TestEnableSTO();

TestPositionMode('Set Target Position_1', 0, 0, 0);
TestPositionMode('Set Target Position_2', 1000, 0, 1000);
TestPositionMode('Set Target Position_3', -1000, 0, -1000);
TestPositionMode('Set Target Position_4', 1000, 100, 1100);
TestPositionMode('Set Target Position_5', 1000, -100, 900);

TestGetProccesData('Get Process Data', FALSE);
TestGetProccesData('Get Process Data Swap', TRUE);
TestSetProccesData('Set Process Data', FALSE);
TestSetProccesData('Set Process Data Swap', TRUE);

METHOD PRIVATE EnableSequence : REFERENCE TO FB_Test
VAR_INPUT
	fbDS402 : REFERENCE TO FB_DS402_CSP;
END_VAR
fbDS402.stControl.nControlWord.b0_SwitchOn := FALSE;
fbDS402.stControl.nControlWord.b1_EnableVoltage := FALSE;
fbDS402.stControl.nControlWord.b2_QuickStop := FALSE;
fbDS402.stControl.nControlWord.b3_EnableOperation := FALSE;
fbDS402();

fbDS402.stControl.nControlWord.b1_EnableVoltage := TRUE;
fbDS402.stControl.nControlWord.b2_QuickStop := TRUE;
fbDS402();
fbDS402.stControl.nControlWord.b0_SwitchOn := TRUE;
fbDS402();
fbDS402.stControl.nControlWord.b3_EnableOperation := TRUE;
fbDS402();
END_METHOD

METHOD TestEnable : BOOL
VAR
	fbDS402 			: FB_DS402_CSP;
	nMask 				: WORD;
	nResult 			: WORD;
	bResult 			: BOOL;
	nActualState		: INT;
	nExpectedState		: INT;
END_VAR
TEST('Enable STO FALSE');
fbDS402.bSTO := FALSE;

EnableSequence(fbDS402);

nExpectedState := E_DS402_State.S0_NotReadyToSwitchOn;
nActualState := fbDS402.eState;

AssertEquals(Expected := nExpectedState,
             Actual := nActualState,
             Message := 'State is not correct');	 
TEST_FINISHED();
END_METHOD

METHOD TestEnableSTO : BOOL
VAR
	fbDS402 			: FB_DS402_CSP;
	nMask 				: WORD;
	nResult 			: WORD;
	bResult 			: BOOL;
	nActualState		: INT;
	nExpectedState		: INT;
END_VAR
TEST('Enable STO TRUE');
fbDS402.bSTO := TRUE;
EnableSequence(fbDS402);

nExpectedState := E_DS402_State.S4_OperationEnabled;
nActualState := fbDS402.eState;

AssertEquals(Expected := nExpectedState,
             Actual := nActualState,
             Message := 'State is not correct');	 
TEST_FINISHED();
END_METHOD

METHOD TestGetProccesData : REFERENCE TO FB_Test
VAR_INPUT
	sName 					: T_MaxString;
	bSwap					: BOOL;
END_VAR

VAR
	fbDS402_CSP 			: FB_DS402_CSP;
	
	aControlData			: ARRAY [0..12] OF BYTE;
	aStatusData				: ARRAY [0..12] OF BYTE;
	
	nControlWordExpected	: WORD; 
	nControlWordActual		: WORD; 
	nTargetExpected			: DINT; 
	nTargetActual			: DINT;	
END_VAR
TEST(sName);

fbDS402_CSP.stConfig.bSwapProcessData := bSwap;
fbDS402_CSP.pControl := ADR(aControlData);
fbDS402_CSP.pStatus := ADR(aStatusData);

nControlWordExpected := 156;
nTargetExpected := 15674;
F_Memcpy(ADR(aControlData), ADR(nControlWordExpected), SIZEOF(nControlWordExpected), bSwap);
F_Memcpy(ADR(aControlData) + 2, ADR(nTargetExpected), SIZEOF(nTargetExpected), bSwap);

fbDS402_CSP.GetControlData();

F_Memcpy(ADR(nControlWordActual), ADR(fbDS402_CSP.stControl.nControlWord), SIZEOF(fbDS402_CSP.stControl.nControlWord), FALSE);
nTargetActual := fbDS402_CSP.stControl.nTargetPosition;

AssertEquals_WORD(Expected := nControlWordExpected,
             Actual := nControlWordActual,
             Message := 'nControlWord is not correct');	

AssertEquals_DINT(Expected := nTargetExpected,
             Actual := nTargetActual,
             Message := '.nTargetPosition is not correct');	

TEST_FINISHED();
END_METHOD

METHOD TestPositionMode : BOOL
VAR_INPUT
	sName 				: T_MaxString;
	fTarget				: LREAL;
	fOffset				: LREAL;
	fExpected			: LREAL;	
END_VAR

VAR
	fbDS402 			: FB_DS402_CSP;	
	fActual 			: LREAL;
	fTolerance 			: LREAL := 1E-6;
END_VAR
TEST(sName);
fbDS402.bSTO := TRUE;
EnableSequence(fbDS402);

fbDS402.stConfig.fPositionOffset := fOffset;
fbDS402.stControl.nTargetPosition := fbDS402.fbEncoder.LREAL_TO_INC(fTarget, 1);

fbDS402();
fActual := fbDS402.fbEncoder.fResult;

AssertEquals_LREAL(Expected := fExpected,
             Actual := fActual,
			 fTolerance,
             Message := 'fbDS402.fbEncoder.fResult is not correct'); 
TEST_FINISHED();
END_METHOD

METHOD TestSetProccesData : REFERENCE TO FB_Test
VAR_INPUT
	sName 					: T_MaxString;
	bSwap					: BOOL;
END_VAR

VAR
	fbDS402_CSP 			: FB_DS402_CSP;
	
	aControlData			: ARRAY [0..12] OF BYTE;
	aStatusData				: ARRAY [0..12] OF BYTE;
	
	nStatusWordExpected		: WORD; 
	nStatusWordActual		: WORD; 
	nActualExpected			: DINT; 
	nActualActual			: DINT;	
	nErrorExpected			: DINT; 
	nErrorActual			: DINT; 
END_VAR
TEST(sName);

fbDS402_CSP.stConfig.bSwapProcessData := bSwap;
fbDS402_CSP.pControl := ADR(aControlData);
fbDS402_CSP.pStatus := ADR(aStatusData);

nStatusWordExpected := 156;
nActualExpected := 15674;
nErrorExpected := 6453;

F_Memcpy(ADR(fbDS402_CSP.stStatus), ADR(nStatusWordExpected), SIZEOF(nStatusWordExpected), FALSE);
F_Memcpy(ADR(fbDS402_CSP.stStatus) + 2, ADR(nActualExpected), SIZEOF(nActualExpected), FALSE);
F_Memcpy(ADR(fbDS402_CSP.stStatus) + 6, ADR(nErrorExpected), SIZEOF(nErrorExpected), FALSE);

fbDS402_CSP.SetStatusData();

F_Memcpy(ADR(nStatusWordActual), ADR(aStatusData), SIZEOF(nStatusWordActual), bSwap);
F_Memcpy(ADR(nActualActual), ADR(aStatusData) + 2, SIZEOF(nActualActual), bSwap);
F_Memcpy(ADR(nErrorActual), ADR(aStatusData) + 6, SIZEOF(nErrorActual), bSwap);


AssertEquals_WORD(Expected := nStatusWordExpected,
             Actual := nStatusWordActual,
             Message := 'nStatusWord is not correct');	

AssertEquals_DINT(Expected := nActualExpected,
             Actual := nActualActual,
             Message := '.nActualPosition is not correct');	
			 
AssertEquals_DINT(Expected := nErrorExpected,
             Actual := nErrorActual,
             Message := '.nErrorActual is not correct');	

TEST_FINISHED();
END_METHOD

END_FUNCTION_BLOCK

// ---- Devices/Drives/DS402/FB_DS402_CSP.TcPOU
(*
	DS402 with Cyclic synchronous position mode(CSP)
	SM2 PDO: 0x1600 (DS402 Controlword)	
	SM2 PDO: 0x1606 (DS402 Target position)
	SM3 PDO: 0x1A00 (DS402 Statusword)	
	SM3 PDO: 0x1A01 (DS402 Position actual value)
	SM3 PDO: 0x1A04 (DS402 Following error actual value)
*)
{attribute 'reflection'} 
FUNCTION_BLOCK FB_DS402_CSP EXTENDS FB_LinkDataReal 
VAR_INPUT
	pControl			: PVOID; //Pocess data from fieldbus, 6 BYTES FROM FIELDBUS
	pStatus				: PVOID; //Pocess data to fieldbus, 6 BYTES FROM FIELDBUS		
	stControl	 		: ST_DS402_CSP_Control;
	stConfig			: ST_DS402_CSP_Config;
	bSTO 				: BOOL := TRUE;
END_VAR

VAR_OUTPUT
	stStatus 			: ST_DS402_CSP_Status;	
END_VAR

VAR		
	{attribute 'instance-path'} 
    {attribute 'noinit'} 
    _sPath 				: STRING;
	_fbStateMachine 	: FB_DS402_FSM;
	_fbEncoder 			: FB_Encoder;	
END_VAR

SUPER^();
InitRun();

GetControlData();
Cycle();
SetStatusData();

METHOD PRIVATE Cycle
IF NOT bSTO THEN RETURN; END_IF

_fbStateMachine.stControl := stControl.nControlWord;
_fbStateMachine();
stStatus.nStatusWord := _fbStateMachine.stStatus;

IF (_fbStateMachine._eState = E_DS402_State.S4_OperationEnabled) THEN	
	
	_fbEncoder.fValue :=  stConfig.fPositionOffset + _fbEncoder.INC_TO_LREAL(stControl.nTargetPosition, 1);
	_fbEncoder();
END_IF

IF stConfig.bSyncOpMode THEN
	stStatus.nStatusWord.b12_OperationModeSpecific := stControl.nControlWord.b4_OperationModeSpecific;
	stStatus.nStatusWord.b13_OperationModeSpecific := stControl.nControlWord.b5_OperationModeSpecific;
	stStatus.nStatusWord.b14_OperationModeSpecific := stControl.nControlWord.b6_OperationModeSpecific;
END_IF


stStatus.nActualPosition := _fbEncoder.nResult;

//Set Link Data
ControlData := LREAL_TO_REAL(_fbEncoder.fResult);
END_METHOD

PROPERTY eState : E_DS402_State
GET
eState := _fbStateMachine.eState;
END_GET
END_PROPERTY

PROPERTY PUBLIC fbEncoder : REFERENCE TO FB_Encoder
GET
fbEncoder REF= _fbEncoder;
END_GET
END_PROPERTY

METHOD INTERNAL GetControlData
IF pControl <= 0 OR stConfig.bForceMode THEN RETURN; END_IF

(*Control Word*)
F_Memcpy(ADR(stControl), pControl, 2, stConfig.bSwapProcessData);
(*Target Value*)
F_Memcpy(ADR(stControl) + 2, pControl + 2, 4, stConfig.bSwapProcessData);
END_METHOD

METHOD PRIVATE InitRun
VAR_INST
	bInitRun : BOOL := TRUE;
END_VAR
IF NOT bInitRun THEN RETURN; END_IF
bInitRun := FALSE;

IF pControl = 0 OR pStatus = 0 THEN
	ADSLOGSTR(ADSLOG_MSGTYPE_WARN, '%s', CONCAT(_sPath, ' PLC IO is not assigned!'));	
END_IF
END_METHOD

METHOD INTERNAL SetStatusData
IF pStatus <= 0 THEN RETURN; END_IF

(*StatusWord*)
F_Memcpy(pStatus, ADR(stStatus), 2, stConfig.bSwapProcessData);
(*Actual Position*)
F_Memcpy(pStatus + 2, ADR(stStatus) + 2, 4, stConfig.bSwapProcessData);
(*Actual Position Error*)
F_Memcpy(pStatus + 6, ADR(stStatus) + 6, 4, stConfig.bSwapProcessData);
END_METHOD

END_FUNCTION_BLOCK

// ---- Tests/Drives/FB_Sercos_FSM_Test.TcPOU
FUNCTION_BLOCK FB_Sercos_FSM_Test EXTENDS TcUnit.FB_TestSuite

TestStateS1();
TestStateS2();
TestStateS3();
TestStateS4();
TestStateS5a();
TestStateS5b();
TestStateS6();
TestStateS7();
TestStateS8();
TestEnableSequence();

METHOD PRIVATE GetEnableCommand : ST_Sercos_ControlWord
GetEnableCommand.b13_Halt := FALSE;
GetEnableCommand.b14_Start := TRUE;
GetEnableCommand.b15_Enable := TRUE;
END_METHOD

METHOD PRIVATE GetEnableHaltCommand : ST_Sercos_ControlWord
GetEnableHaltCommand.b13_Halt := TRUE;
GetEnableHaltCommand.b14_Start := TRUE;
GetEnableHaltCommand.b15_Enable := TRUE;
END_METHOD

METHOD PRIVATE GetErrorResetCommand : ST_Sercos_ControlWord
GetErrorResetCommand.b13_Halt := TRUE;
END_METHOD

METHOD PRIVATE GetHaltCommand : ST_Sercos_ControlWord
GetHaltCommand.b13_Halt := FALSE;
GetHaltCommand.b14_Start := TRUE;
GetHaltCommand.b15_Enable := TRUE;
END_METHOD

METHOD PRIVATE GetQuickStopCommand : ST_Sercos_ControlWord
GetQuickStopCommand.b14_Start := FALSE;
GetQuickStopCommand.b15_Enable := TRUE;
END_METHOD

METHOD PRIVATE GetRunCommand : ST_Sercos_ControlWord
GetRunCommand.b13_Halt := FALSE;
GetRunCommand.b14_Start := TRUE;
GetRunCommand.b15_Enable := TRUE;
END_METHOD

METHOD PRIVATE GetShutdownCommand : ST_Sercos_ControlWord
GetShutdownCommand.b15_Enable := FALSE;
END_METHOD

METHOD PRIVATE GetSwitchOnCommand : ST_Sercos_ControlWord
GetSwitchOnCommand.b15_Enable := TRUE;
END_METHOD

METHOD TestEnableSequence : BOOL
VAR
	fbSercosFSM 			: FB_Sercos_FSM;
	stExpectedStatus 		: ST_Sercos_StatusWord; 
	nMask 					: WORD;
	nResult 				: WORD;
	bResult 				: BOOL;
	nActualState			: INT;
	nExpectedState			: INT;
END_VAR
TEST('Enable S1');

nExpectedState := E_Sercos_State.S1_NotReadyToSwitchOn;
nActualState := fbSercosFSM.eState;

AssertEquals(Expected := nExpectedState,
             Actual := nActualState,
             Message := 'State is not correct');	 
TEST_FINISHED();

TEST('Enable S2');
fbSercosFSM();
nExpectedState := E_Sercos_State.S2_SwitchOnDisabled;
nActualState := fbSercosFSM.eState;

AssertEquals(Expected := nExpectedState,
             Actual := nActualState,
             Message := 'State is not correct');	 
TEST_FINISHED();

TEST('Enable S3');
fbSercosFSM.bPower := TRUE;
fbSercosFSM();
nExpectedState := E_Sercos_State.S3_ReadyToSwitchOn;
nActualState := fbSercosFSM.eState;

AssertEquals(Expected := nExpectedState,
             Actual := nActualState,
             Message := 'State is not correct');	 
TEST_FINISHED();

TEST('Enable S4');
fbSercosFSM.stControl := GetSwitchOnCommand();

fbSercosFSM();
nExpectedState := E_Sercos_State.S4_SwitchOn;
nActualState := fbSercosFSM.eState;

AssertEquals(Expected := nExpectedState,
             Actual := nActualState,
             Message := 'State is not correct');	 
TEST_FINISHED();

TEST('Enable S5a');
fbSercosFSM.stControl := GetEnableCommand();

fbSercosFSM();
nExpectedState := E_Sercos_State.S5a_DriveInOperation;
nActualState := fbSercosFSM.eState;

AssertEquals(Expected := nExpectedState,
             Actual := nActualState,
             Message := 'State is not correct');	 
TEST_FINISHED();
END_METHOD

METHOD TestStateS1 : BOOL
VAR
	fbSercosFSM 		: FB_Sercos_FSM;
	stExpectedStatus 	: ST_Sercos_StatusWord; 
	nMask 				: WORD;
	nResult 			: WORD;
	bResult 			: BOOL;
	nActualState		: INT;
	nExpectedState		: INT;
END_VAR
TEST('Set State S1');
fbSercosFSM.eState := E_Sercos_State.S1_NotReadyToSwitchOn;
fbSercosFSM();

stExpectedStatus.b15_ReadyToOperate 		:= FALSE;
stExpectedStatus.b14_ReadyToOperate 		:= FALSE;
stExpectedStatus.b13_Error 					:= FALSE;
stExpectedStatus.b7_QuickStop 				:= FALSE;
stExpectedStatus.b4_Halt 					:= FALSE;
stExpectedStatus.b3_CommandProcessing 		:= FALSE;

MEMCPY(ADR(nMask), ADR(stExpectedStatus), 2);
nResult := (2#1110000011011000 AND fbSercosFSM.nStatus);

AssertEquals(Expected := nMask,
             Actual := nResult,
             Message := 'Value is not correct');	 
TEST_FINISHED();

TEST('Transition S1>S2');
fbSercosFSM.eState := E_Sercos_State.S1_NotReadyToSwitchOn;
fbSercosFSM();

nExpectedState := E_Sercos_State.S2_SwitchOnDisabled;
nActualState := fbSercosFSM.eState;

AssertEquals(Expected := nExpectedState,
             Actual := nActualState,
             Message := 'State is not correct');	 
TEST_FINISHED();
END_METHOD

METHOD TestStateS2 : BOOL
VAR
	fbSercosFSM 		: FB_Sercos_FSM;
	stExpectedStatus 	: ST_Sercos_StatusWord; 
	nMask 				: WORD;
	nResult 			: WORD;
	bResult 			: BOOL;
	nActualState		: INT;
	nExpectedState		: INT;
END_VAR
TEST('Set State S2');
fbSercosFSM.eState := E_Sercos_State.S2_SwitchOnDisabled;
fbSercosFSM();

stExpectedStatus.b15_ReadyToOperate 		:= FALSE;
stExpectedStatus.b14_ReadyToOperate 		:= TRUE;
stExpectedStatus.b13_Error 					:= FALSE;
stExpectedStatus.b7_QuickStop 				:= FALSE;
stExpectedStatus.b4_Halt 					:= FALSE;
stExpectedStatus.b3_CommandProcessing 		:= FALSE;

MEMCPY(ADR(nMask), ADR(stExpectedStatus), 2);
nResult := (2#1110000011011000 AND fbSercosFSM.nStatus);

AssertEquals(Expected := nMask,
             Actual := nResult,
             Message := 'Value is not correct');	 
TEST_FINISHED();

TEST('Still State S2');
fbSercosFSM.bPower := FALSE;
fbSercosFSM.eState := E_Sercos_State.S2_SwitchOnDisabled;
fbSercosFSM();

nExpectedState := E_Sercos_State.S2_SwitchOnDisabled;
nActualState := fbSercosFSM.eState;

AssertEquals(Expected := nExpectedState,
             Actual := nActualState,
             Message := 'State is not correct');	 
TEST_FINISHED();

TEST('Transition S2>S3');
fbSercosFSM.bPower := TRUE;
fbSercosFSM.eState := E_Sercos_State.S2_SwitchOnDisabled;
fbSercosFSM();

nExpectedState := E_Sercos_State.S3_ReadyToSwitchOn;
nActualState := fbSercosFSM.eState;

AssertEquals(Expected := nExpectedState,
             Actual := nActualState,
             Message := 'State is not correct');	 
TEST_FINISHED();
END_METHOD

METHOD TestStateS3 : BOOL
VAR
	fbSercosFSM 		: FB_Sercos_FSM;
	stExpectedStatus 	: ST_Sercos_StatusWord; 
	nMask 				: WORD;
	nResult 			: WORD;
	bResult 			: BOOL;
	nActualState		: INT;
	nExpectedState		: INT;
END_VAR
TEST('Set State S3');
fbSercosFSM.eState := E_Sercos_State.S3_ReadyToSwitchOn;
fbSercosFSM();

stExpectedStatus.b15_ReadyToOperate 		:= TRUE;
stExpectedStatus.b14_ReadyToOperate 		:= FALSE;
stExpectedStatus.b13_Error 					:= FALSE;
stExpectedStatus.b7_QuickStop 				:= FALSE;
stExpectedStatus.b4_Halt 					:= FALSE;
stExpectedStatus.b3_CommandProcessing 		:= FALSE;

MEMCPY(ADR(nMask), ADR(stExpectedStatus), 2);
nResult := (2#1110000011011000 AND fbSercosFSM.nStatus);

AssertEquals(Expected := nMask,
             Actual := nResult,
             Message := 'Value is not correct');	 
TEST_FINISHED();

TEST('Transition S3>S2');
fbSercosFSM.bPower := FALSE;
fbSercosFSM.eState := E_Sercos_State.S3_ReadyToSwitchOn;
fbSercosFSM();

nExpectedState := E_Sercos_State.S2_SwitchOnDisabled;
nActualState := fbSercosFSM.eState;

AssertEquals(Expected := nExpectedState,
             Actual := nActualState,
             Message := 'State is not correct');	 
TEST_FINISHED();

TEST('Transition S3>S7');
fbSercosFSM.bPower := TRUE;
fbSercosFSM.bError := TRUE;
fbSercosFSM.eState := E_Sercos_State.S3_ReadyToSwitchOn;
fbSercosFSM();

nExpectedState := E_Sercos_State.S7_FaultReactionActive;
nActualState := fbSercosFSM.eState;

AssertEquals(Expected := nExpectedState,
             Actual := nActualState,
             Message := 'State is not correct');	 
TEST_FINISHED();

TEST('Transition S3>S4');
fbSercosFSM.bError := FALSE;
fbSercosFSM.stControl := GetSwitchOnCommand();
fbSercosFSM.eState := E_Sercos_State.S3_ReadyToSwitchOn;
fbSercosFSM();

nExpectedState := E_Sercos_State.S4_SwitchOn;
nActualState := fbSercosFSM.eState;

AssertEquals(Expected := nExpectedState,
             Actual := nActualState,
             Message := 'State is not correct');	 
TEST_FINISHED();
END_METHOD

METHOD TestStateS4 : BOOL
VAR
	fbSercosFSM 		: FB_Sercos_FSM;
	stExpectedStatus 	: ST_Sercos_StatusWord; 
	nMask 				: WORD;
	nResult 			: WORD;
	bResult 			: BOOL;
	nActualState		: INT;
	nExpectedState		: INT;
END_VAR
TEST('Set State S4');
fbSercosFSM.eState := E_Sercos_State.S4_SwitchOn;
fbSercosFSM();

stExpectedStatus.b15_ReadyToOperate 		:= FALSE;
stExpectedStatus.b14_ReadyToOperate 		:= TRUE;
stExpectedStatus.b13_Error 					:= FALSE;
stExpectedStatus.b7_QuickStop 				:= FALSE;
stExpectedStatus.b4_Halt 					:= FALSE;
stExpectedStatus.b3_CommandProcessing 		:= FALSE;

MEMCPY(ADR(nMask), ADR(stExpectedStatus), 2);
nResult := (2#1110000011011000 AND fbSercosFSM.nStatus);

AssertEquals(Expected := nMask,
             Actual := nResult,
             Message := 'Value is not correct');	 
TEST_FINISHED();

TEST('Transition S4>S2');
fbSercosFSM.bPower := FALSE;
fbSercosFSM.eState := E_Sercos_State.S4_SwitchOn;
fbSercosFSM();
fbSercosFSM();

nExpectedState := E_Sercos_State.S2_SwitchOnDisabled;
nActualState := fbSercosFSM.eState;

AssertEquals(Expected := nExpectedState,
             Actual := nActualState,
             Message := 'State is not correct');	 
TEST_FINISHED();

TEST('Transition S4>S3');
fbSercosFSM.bPower := TRUE;
fbSercosFSM.eState := E_Sercos_State.S4_SwitchOn;
fbSercosFSM.stControl := GetShutdownCommand();
fbSercosFSM();

nExpectedState := E_Sercos_State.S3_ReadyToSwitchOn;
nActualState := fbSercosFSM.eState;

AssertEquals(Expected := nExpectedState,
             Actual := nActualState,
             Message := 'State is not correct');	 
TEST_FINISHED();

TEST('Transition S4>S7');
fbSercosFSM.bPower := TRUE;
fbSercosFSM.bError := TRUE;
fbSercosFSM.eState := E_Sercos_State.S4_SwitchOn;
fbSercosFSM();

nExpectedState := E_Sercos_State.S7_FaultReactionActive;
nActualState := fbSercosFSM.eState;

AssertEquals(Expected := nExpectedState,
             Actual := nActualState,
             Message := 'State is not correct');	 
TEST_FINISHED();

TEST('Transition S4>S5b');
fbSercosFSM.bError := FALSE;
fbSercosFSM.stControl := GetEnableHaltCommand();
fbSercosFSM.eState := E_Sercos_State.S4_SwitchOn;
fbSercosFSM();

nExpectedState := E_Sercos_State.S5b_Halt;
nActualState := fbSercosFSM.eState;

AssertEquals(Expected := nExpectedState,
             Actual := nActualState,
             Message := 'State is not correct');	 
TEST_FINISHED();

TEST('Transition S4>S5a');
fbSercosFSM.bError := FALSE;
fbSercosFSM.stControl := GetEnableCommand();
fbSercosFSM.eState := E_Sercos_State.S4_SwitchOn;
fbSercosFSM();

nExpectedState := E_Sercos_State.S5a_DriveInOperation;
nActualState := fbSercosFSM.eState;

AssertEquals(Expected := nExpectedState,
             Actual := nActualState,
             Message := 'State is not correct');	 
TEST_FINISHED();
END_METHOD

METHOD TestStateS5a : BOOL
VAR
	fbSercosFSM 		: FB_Sercos_FSM;
	stExpectedStatus 	: ST_Sercos_StatusWord; 
	nMask 				: WORD;
	nResult 			: WORD;
	bResult 			: BOOL;
	nActualState		: INT;
	nExpectedState		: INT;
END_VAR
TEST('Set State S5a');
fbSercosFSM.eState := E_Sercos_State.S5a_DriveInOperation;
fbSercosFSM();

stExpectedStatus.b15_ReadyToOperate 		:= TRUE;
stExpectedStatus.b14_ReadyToOperate 		:= TRUE;
stExpectedStatus.b13_Error 					:= FALSE;
stExpectedStatus.b7_QuickStop 				:= FALSE;
stExpectedStatus.b4_Halt 					:= FALSE;
stExpectedStatus.b3_CommandProcessing 		:= TRUE;

MEMCPY(ADR(nMask), ADR(stExpectedStatus), 2);
nResult := (2#1110000011011000 AND fbSercosFSM.nStatus);

AssertEquals(Expected := nMask,
             Actual := nResult,
             Message := 'Value is not correct');	 
TEST_FINISHED();

TEST('Transition S5a>S2');
fbSercosFSM.bPower := FALSE;
fbSercosFSM.eState := E_Sercos_State.S5a_DriveInOperation;
fbSercosFSM();
fbSercosFSM();

nExpectedState := E_Sercos_State.S2_SwitchOnDisabled;
nActualState := fbSercosFSM.eState;

AssertEquals(Expected := nExpectedState,
             Actual := nActualState,
             Message := 'State is not correct');	 
TEST_FINISHED();

TEST('Transition S5a>S7');
fbSercosFSM.bPower := TRUE;
fbSercosFSM.bError := TRUE;
fbSercosFSM.eState := E_Sercos_State.S5a_DriveInOperation;
fbSercosFSM();

nExpectedState := E_Sercos_State.S7_FaultReactionActive;
nActualState := fbSercosFSM.eState;

AssertEquals(Expected := nExpectedState,
             Actual := nActualState,
             Message := 'State is not correct');	 
TEST_FINISHED();

TEST('Transition S5a>S3');
fbSercosFSM.bError := FALSE;
fbSercosFSM.bPower := TRUE;
fbSercosFSM.eState := E_Sercos_State.S5a_DriveInOperation;
fbSercosFSM.stControl := GetShutdownCommand();
fbSercosFSM();

nExpectedState := E_Sercos_State.S3_ReadyToSwitchOn;
nActualState := fbSercosFSM.eState;

AssertEquals(Expected := nExpectedState,
             Actual := nActualState,
             Message := 'State is not correct');	 
TEST_FINISHED();

TEST('Transition S5a>S6');
fbSercosFSM.bError := FALSE;
fbSercosFSM.bPower := TRUE;
fbSercosFSM.eState := E_Sercos_State.S5a_DriveInOperation;
fbSercosFSM.stControl := GetQuickStopCommand();
fbSercosFSM();

nExpectedState := E_Sercos_State.S6_QuickStop;
nActualState := fbSercosFSM.eState;

AssertEquals(Expected := nExpectedState,
             Actual := nActualState,
             Message := 'State is not correct');	 
TEST_FINISHED();

TEST('Transition S5a>S5b');
fbSercosFSM.bError := FALSE;
fbSercosFSM.bPower := TRUE;
fbSercosFSM.stControl := GetEnableHaltCommand();
fbSercosFSM.eState := E_Sercos_State.S5a_DriveInOperation;
fbSercosFSM();

nExpectedState := E_Sercos_State.S5b_Halt;
nActualState := fbSercosFSM.eState;

AssertEquals(Expected := nExpectedState,
             Actual := nActualState,
             Message := 'State is not correct');	 
TEST_FINISHED();
END_METHOD

METHOD TestStateS5b : BOOL
VAR
	fbSercosFSM 		: FB_Sercos_FSM;
	stExpectedStatus 	: ST_Sercos_StatusWord; 
	nMask 				: WORD;
	nResult 			: WORD;
	bResult 			: BOOL;
	nActualState		: INT;
	nExpectedState		: INT;
END_VAR
TEST('Set State S5b');
fbSercosFSM.eState := E_Sercos_State.S5b_Halt;
fbSercosFSM();

stExpectedStatus.b15_ReadyToOperate 		:= TRUE;
stExpectedStatus.b14_ReadyToOperate 		:= TRUE;
stExpectedStatus.b13_Error 					:= FALSE;
stExpectedStatus.b7_QuickStop 				:= FALSE;
stExpectedStatus.b4_Halt 					:= TRUE;
stExpectedStatus.b3_CommandProcessing 		:= FALSE;

MEMCPY(ADR(nMask), ADR(stExpectedStatus), 2);
nResult := (2#1110000011011000 AND fbSercosFSM.nStatus);

AssertEquals(Expected := nMask,
             Actual := nResult,
             Message := 'Value is not correct');	 
TEST_FINISHED();

TEST('Transition S5b>S2');
fbSercosFSM.bPower := FALSE;
fbSercosFSM.eState := E_Sercos_State.S5b_Halt;
fbSercosFSM();

nExpectedState := E_Sercos_State.S2_SwitchOnDisabled;
nActualState := fbSercosFSM.eState;

AssertEquals(Expected := nExpectedState,
             Actual := nActualState,
             Message := 'State is not correct');	 
TEST_FINISHED();

TEST('Transition S5b>S7');
fbSercosFSM.bPower := TRUE;
fbSercosFSM.bError := TRUE;
fbSercosFSM.eState := E_Sercos_State.S5b_Halt;
fbSercosFSM();

nExpectedState := E_Sercos_State.S7_FaultReactionActive;
nActualState := fbSercosFSM.eState;

AssertEquals(Expected := nExpectedState,
             Actual := nActualState,
             Message := 'State is not correct');	 
TEST_FINISHED();

TEST('Transition S5b>S3');
fbSercosFSM.bError := FALSE;
fbSercosFSM.bPower := TRUE;
fbSercosFSM.eState := E_Sercos_State.S5b_Halt;
fbSercosFSM.stControl := GetShutdownCommand();
fbSercosFSM();

nExpectedState := E_Sercos_State.S3_ReadyToSwitchOn;
nActualState := fbSercosFSM.eState;

AssertEquals(Expected := nExpectedState,
             Actual := nActualState,
             Message := 'State is not correct');	 
TEST_FINISHED();

TEST('Transition S5b>S6');
fbSercosFSM.bError := FALSE;
fbSercosFSM.bPower := TRUE;
fbSercosFSM.eState := E_Sercos_State.S5b_Halt;
fbSercosFSM.stControl := GetQuickStopCommand();
fbSercosFSM();

nExpectedState := E_Sercos_State.S6_QuickStop;
nActualState := fbSercosFSM.eState;

AssertEquals(Expected := nExpectedState,
             Actual := nActualState,
             Message := 'State is not correct');	 
TEST_FINISHED();

TEST('Transition S5b>S5a');
fbSercosFSM.bError := FALSE;
fbSercosFSM.bPower := TRUE;
fbSercosFSM.stControl := GetEnableCommand();
fbSercosFSM.eState := E_Sercos_State.S5b_Halt;
fbSercosFSM();

nExpectedState := E_Sercos_State.S5a_DriveInOperation;
nActualState := fbSercosFSM.eState;

AssertEquals(Expected := nExpectedState,
             Actual := nActualState,
             Message := 'State is not correct');	 
TEST_FINISHED();
END_METHOD

METHOD TestStateS6 : BOOL
VAR
	fbSercosFSM 		: FB_Sercos_FSM;
	stExpectedStatus 	: ST_Sercos_StatusWord; 
	nMask 				: WORD;
	nResult 			: WORD;
	bResult 			: BOOL;
	nActualState		: INT;
	nExpectedState		: INT;
END_VAR
TEST('Set State S6');
fbSercosFSM.eState := E_Sercos_State.S6_QuickStop;
fbSercosFSM();

stExpectedStatus.b15_ReadyToOperate 		:= TRUE;
stExpectedStatus.b14_ReadyToOperate 		:= TRUE;
stExpectedStatus.b13_Error 					:= FALSE;
stExpectedStatus.b7_QuickStop 				:= TRUE;
stExpectedStatus.b4_Halt 					:= TRUE;
stExpectedStatus.b3_CommandProcessing 		:= FALSE;

MEMCPY(ADR(nMask), ADR(stExpectedStatus), 2);
nResult := (2#1110000011011000 AND fbSercosFSM.nStatus);

AssertEquals(Expected := nMask,
             Actual := nResult,
             Message := 'Value is not correct');	 
TEST_FINISHED();

TEST('Transition S6>S2');
fbSercosFSM.bPower := FALSE;
fbSercosFSM.eState := E_Sercos_State.S6_QuickStop;
fbSercosFSM();
fbSercosFSM();

nExpectedState := E_Sercos_State.S2_SwitchOnDisabled;
nActualState := fbSercosFSM.eState;

AssertEquals(Expected := nExpectedState,
             Actual := nActualState,
             Message := 'State is not correct');	 
TEST_FINISHED();

TEST('Transition S6>S3');
fbSercosFSM.bPower := TRUE;
fbSercosFSM.eState := E_Sercos_State.S6_QuickStop;
fbSercosFSM.stControl := GetShutdownCommand();
fbSercosFSM();

nExpectedState := E_Sercos_State.S3_ReadyToSwitchOn;
nActualState := fbSercosFSM.eState;

AssertEquals(Expected := nExpectedState,
             Actual := nActualState,
             Message := 'State is not correct');	 
TEST_FINISHED();

TEST('Transition S6>S7');
fbSercosFSM.bPower := TRUE;
fbSercosFSM.bError := TRUE;
fbSercosFSM.eState := E_Sercos_State.S6_QuickStop;
fbSercosFSM();

nExpectedState := E_Sercos_State.S7_FaultReactionActive;
nActualState := fbSercosFSM.eState;

AssertEquals(Expected := nExpectedState,
             Actual := nActualState,
             Message := 'State is not correct');	 
TEST_FINISHED();

TEST('Transition S6>S5b');
fbSercosFSM.bError := FALSE;
fbSercosFSM.stControl := GetEnableHaltCommand();
fbSercosFSM.eState := E_Sercos_State.S6_QuickStop;
fbSercosFSM();

nExpectedState := E_Sercos_State.S5b_Halt;
nActualState := fbSercosFSM.eState;

AssertEquals(Expected := nExpectedState,
             Actual := nActualState,
             Message := 'State is not correct');	 
TEST_FINISHED();

TEST('Transition S6>S5a');
fbSercosFSM.bError := FALSE;
fbSercosFSM.stControl := GetEnableCommand();
fbSercosFSM.eState := E_Sercos_State.S6_QuickStop;
fbSercosFSM();

nExpectedState := E_Sercos_State.S5a_DriveInOperation;
nActualState := fbSercosFSM.eState;

AssertEquals(Expected := nExpectedState,
             Actual := nActualState,
             Message := 'State is not correct');	 
TEST_FINISHED();
END_METHOD

METHOD TestStateS7 : BOOL
VAR
	fbSercosFSM 		: FB_Sercos_FSM;
	stExpectedStatus 	: ST_Sercos_StatusWord; 
	nMask 				: WORD;
	nResult 			: WORD;
	bResult 			: BOOL;
	nActualState		: INT;
	nExpectedState		: INT;
END_VAR
TEST('Set State S7');
fbSercosFSM.eState := E_Sercos_State.S7_FaultReactionActive;
fbSercosFSM();

stExpectedStatus.b15_ReadyToOperate 		:= TRUE;
stExpectedStatus.b14_ReadyToOperate 		:= TRUE;
stExpectedStatus.b13_Error 					:= TRUE;
stExpectedStatus.b7_QuickStop 				:= FALSE;
stExpectedStatus.b4_Halt 					:= FALSE;
stExpectedStatus.b3_CommandProcessing 		:= FALSE;

MEMCPY(ADR(nMask), ADR(stExpectedStatus), 2);
nResult := (2#1110000011011000 AND fbSercosFSM.nStatus);

AssertEquals(Expected := nMask,
             Actual := nResult,
             Message := 'Value is not correct');	 
TEST_FINISHED();

TEST('Transition S7>S2');
fbSercosFSM.bPower := FALSE;
fbSercosFSM.eState := E_Sercos_State.S7_FaultReactionActive;
fbSercosFSM();

nExpectedState := E_Sercos_State.S2_SwitchOnDisabled;
nActualState := fbSercosFSM.eState;

AssertEquals(Expected := nExpectedState,
             Actual := nActualState,
             Message := 'State is not correct');	 
TEST_FINISHED();

TEST('Transition S7>S8');
fbSercosFSM.bPower := TRUE;
fbSercosFSM.eState := E_Sercos_State.S7_FaultReactionActive;
fbSercosFSM();

nExpectedState := E_Sercos_State.S8_Fault;
nActualState := fbSercosFSM.eState;

AssertEquals(Expected := nExpectedState,
             Actual := nActualState,
             Message := 'State is not correct');	 
TEST_FINISHED();
END_METHOD

METHOD TestStateS8 : BOOL
VAR
	fbSercosFSM 		: FB_Sercos_FSM;
	stExpectedStatus 	: ST_Sercos_StatusWord; 
	nMask 				: WORD;
	nResult 			: WORD;
	bResult 			: BOOL;
	nActualState		: INT;
	nExpectedState		: INT;
END_VAR
TEST('Set State S8');
fbSercosFSM.eState := E_Sercos_State.S8_Fault;
fbSercosFSM();

stExpectedStatus.b15_ReadyToOperate 		:= TRUE;
stExpectedStatus.b14_ReadyToOperate 		:= FALSE;
stExpectedStatus.b13_Error 					:= TRUE;
stExpectedStatus.b7_QuickStop 				:= FALSE;
stExpectedStatus.b4_Halt 					:= FALSE;
stExpectedStatus.b3_CommandProcessing 		:= FALSE;

MEMCPY(ADR(nMask), ADR(stExpectedStatus), 2);
nResult := (2#1110000011011000 AND fbSercosFSM.nStatus);

AssertEquals(Expected := nMask,
             Actual := nResult,
             Message := 'Value is not correct');	 
TEST_FINISHED();

TEST('Transition S8>S2');
fbSercosFSM.bPower := FALSE;
fbSercosFSM.eState := E_Sercos_State.S8_Fault;
fbSercosFSM.stControl := GetErrorResetCommand();
fbSercosFSM();

nExpectedState := E_Sercos_State.S2_SwitchOnDisabled;
nActualState := fbSercosFSM.eState;

AssertEquals(Expected := nExpectedState,
             Actual := nActualState,
             Message := 'State is not correct');	 
TEST_FINISHED();
END_METHOD

END_FUNCTION_BLOCK

// ---- Devices/Drives/Sercos/FB_Sercos_FSM.TcPOU
(*
	Sercos Finite State Machine General
*)
FUNCTION_BLOCK FB_Sercos_FSM
VAR_INPUT
	bPower						: BOOL := TRUE;	
	stControl					: ST_Sercos_ControlWord;
END_VAR

VAR_OUTPUT	
	stStatus					: ST_Sercos_StatusWord;	
END_VAR

VAR	
	_eState 					: E_Sercos_State := E_Sercos_State.S1_NotReadyToSwitchOn;
	_rTrig_Reset 				: R_TRIG;
	_bError						: BOOL;
END_VAR

_rTrig_Reset(CLK := stControl.b13_Halt);

CASE _eState OF
	E_Sercos_State.S1_NotReadyToSwitchOn 	: S1_NotReadyToSwitchOn();
	E_Sercos_State.S2_SwitchOnDisabled 		: S2_SwitchOnDisabled();
	E_Sercos_State.S3_ReadyToSwitchOn 		: S3_ReadyToSwitchOn();
	E_Sercos_State.S4_SwitchOn 				: S4_SwitchOn();
	E_Sercos_State.S5a_DriveInOperation 	: S5a_DriveInOperation();
	E_Sercos_State.S5b_Halt 				: S5b_Halt();	
	E_Sercos_State.S6_QuickStop 			: S6_QuickStop();	
	E_Sercos_State.S7_FaultReactionActive 	: S7_FaultReactionActive();
	E_Sercos_State.S8_Fault 				: S8_Fault();
END_CASE

PROPERTY PUBLIC bError : BOOL
GET
bError := _bError;
END_GET
SET
_bError := bError;
END_SET
END_PROPERTY

PROPERTY eState : E_Sercos_State
GET
eState := _eState;
END_GET
SET
_eState := eState;
END_SET
END_PROPERTY

PROPERTY nControl : WORD
GET
nControl.0	:= stControl.b0_Reserved;					           
nControl.1	:= stControl.b1_Reserved;						        	
nControl.2	:= stControl.b2_Reserved;						           	
nControl.3	:= stControl.b3_Reserved;						       	
nControl.4	:= stControl.b4_Reserved;						    
nControl.5	:= stControl.b5_Reserved;						    
nControl.6	:= stControl.b6_Reserved;						    
nControl.7	:= stControl.b7_Reserved;						          	
nControl.8	:= stControl.b8_Reserved;						            	
nControl.9	:= stControl.b9_Reserved;						            
nControl.10	:= stControl.b10_OperationMode;				       	
nControl.11	:= stControl.b11_Reserved;					           	
nControl.12	:= stControl.b12_Reserved;
nControl.13	:= stControl.b13_Halt;						              	
nControl.14	:= stControl.b14_Start;						            	
nControl.15 := stControl.b15_Enable;
END_GET
SET
stControl.b0_Reserved 					:= 	nControl.0;	
stControl.b1_Reserved					:= 	nControl.1;		
stControl.b2_Reserved					:= 	nControl.2;		
stControl.b3_Reserved					:= 	nControl.3;		
stControl.b4_Reserved					:= 	nControl.4;		
stControl.b5_Reserved					:= 	nControl.5;		
stControl.b6_Reserved					:= 	nControl.6;		
stControl.b7_Reserved					:= 	nControl.7;		
stControl.b8_Reserved					:= 	nControl.8;		
stControl.b9_Reserved					:= 	nControl.9;		
stControl.b10_OperationMode				:= 	nControl.10;		
stControl.b11_Reserved					:= 	nControl.11;		
stControl.b12_Reserved					:= 	nControl.12;		
stControl.b13_Halt						:= 	nControl.13;		
stControl.b14_Start					:= 	nControl.14;		
stControl.b15_Enable						:= 	nControl.15;
END_SET
END_PROPERTY

PROPERTY nStatus : WORD
GET
nStatus.0 	:= stStatus.b0_Reserved;					      
nStatus.1 	:= stStatus.b1_Reserved;						      
nStatus.2 	:= stStatus.b2_Reserved;						      
nStatus.3 	:= stStatus.b3_CommandProcessing;		
nStatus.4 	:= stStatus.b4_Halt;							         
nStatus.5 	:= stStatus.b5_PositionFeedback;		
nStatus.6 	:= stStatus.b6_Reserved;					      
nStatus.7 	:= stStatus.b7_QuickStop;					      
nStatus.8 	:= stStatus.b8_Reserved;					      
nStatus.9 	:= stStatus.b9_Reserved;					      
nStatus.10 	:= stStatus.b10_OperationMode;		  
nStatus.11 	:= stStatus.b11_Reserved;					      
nStatus.12 	:= stStatus.b12_Warning;					      
nStatus.13 	:= stStatus.b13_Error;					        
nStatus.14 	:= stStatus.b14_ReadyToOperate;			 
nStatus.15 	:= stStatus.b15_ReadyToOperate;
END_GET
END_PROPERTY

METHOD PRIVATE S1_NotReadyToSwitchOn : BOOL
VAR_INPUT
END_VAR
stStatus.b15_ReadyToOperate 		:= FALSE;
stStatus.b14_ReadyToOperate 		:= FALSE;
stStatus.b13_Error 					:= FALSE;
stStatus.b7_QuickStop 				:= FALSE;
stStatus.b4_Halt 					:= FALSE;
stStatus.b3_CommandProcessing 		:= FALSE;

_eState := E_Sercos_State.S2_SwitchOnDisabled;
END_METHOD

METHOD PRIVATE S2_SwitchOnDisabled : BOOL
VAR_INPUT
END_VAR
stStatus.b15_ReadyToOperate 		:= FALSE;
stStatus.b14_ReadyToOperate 		:= TRUE;
stStatus.b13_Error 					:= FALSE;
stStatus.b7_QuickStop 				:= FALSE;
stStatus.b4_Halt 					:= FALSE;
stStatus.b3_CommandProcessing 		:= FALSE;

IF bPower THEN
	_eState := E_Sercos_State.S3_ReadyToSwitchOn;
	RETURN;
END_IF
END_METHOD

METHOD PRIVATE S3_ReadyToSwitchOn : BOOL
VAR_INPUT
END_VAR
stStatus.b15_ReadyToOperate 		:= TRUE;
stStatus.b14_ReadyToOperate 		:= FALSE;
stStatus.b13_Error 					:= FALSE;
stStatus.b7_QuickStop 				:= FALSE;
stStatus.b4_Halt 					:= FALSE;
stStatus.b3_CommandProcessing 		:= FALSE;

IF NOT bPower THEN
	_eState := E_Sercos_State.S2_SwitchOnDisabled;
	RETURN;
END_IF

IF _bError THEN
	_eState := E_Sercos_State.S7_FaultReactionActive;
	RETURN;
END_IF

IF stControl.b15_Enable THEN
	_eState := E_Sercos_State.S4_SwitchOn;
	RETURN;
END_IF
END_METHOD

METHOD PRIVATE S4_SwitchOn : BOOL
VAR_INPUT
END_VAR
stStatus.b15_ReadyToOperate 		:= FALSE;
stStatus.b14_ReadyToOperate 		:= TRUE;
stStatus.b13_Error 					:= FALSE;
stStatus.b7_QuickStop 				:= FALSE;
stStatus.b4_Halt 					:= FALSE;
stStatus.b3_CommandProcessing 		:= FALSE;

IF NOT bPower THEN
	_eState := E_Sercos_State.S2_SwitchOnDisabled;
	RETURN;
END_IF

IF _bError THEN
	_eState := E_Sercos_State.S7_FaultReactionActive;
	RETURN;
END_IF

IF NOT stControl.b15_Enable THEN 
	_eState := E_Sercos_State.S3_ReadyToSwitchOn;
	RETURN;
END_IF

IF stControl.b13_Halt AND stControl.b14_Start THEN
	_eState := E_Sercos_State.S5b_Halt;
	RETURN;
END_IF

IF NOT stControl.b13_Halt AND stControl.b14_Start THEN
	_eState := E_Sercos_State.S5a_DriveInOperation;
	RETURN;
END_IF
END_METHOD

METHOD PRIVATE S5a_DriveInOperation : BOOL
VAR_INPUT
END_VAR
stStatus.b15_ReadyToOperate 		:= TRUE;
stStatus.b14_ReadyToOperate 		:= TRUE;
stStatus.b13_Error 					:= FALSE;
stStatus.b7_QuickStop 				:= FALSE;
stStatus.b4_Halt 					:= FALSE;
stStatus.b3_CommandProcessing 		:= TRUE;

IF NOT bPower THEN
	_eState := E_Sercos_State.S2_SwitchOnDisabled;
	RETURN;
END_IF

IF _bError THEN
	_eState := E_Sercos_State.S7_FaultReactionActive;
	RETURN;
END_IF

IF NOT stControl.b15_Enable THEN 
	_eState := E_Sercos_State.S3_ReadyToSwitchOn;
	RETURN;
END_IF

IF NOT stControl.b14_Start THEN
	_eState := E_Sercos_State.S6_QuickStop;
	RETURN;
END_IF

IF stControl.b13_Halt THEN
	_eState := E_Sercos_State.S5b_Halt;
	RETURN;
END_IF
END_METHOD

METHOD PRIVATE S5b_Halt : BOOL
VAR_INPUT
END_VAR
stStatus.b15_ReadyToOperate 		:= TRUE;
stStatus.b14_ReadyToOperate 		:= TRUE;
stStatus.b13_Error 					:= FALSE;
stStatus.b7_QuickStop 				:= FALSE;
stStatus.b4_Halt 					:= TRUE;
stStatus.b3_CommandProcessing 		:= FALSE;

IF NOT bPower THEN
	_eState := E_Sercos_State.S2_SwitchOnDisabled;
	RETURN;
END_IF

IF _bError THEN
	_eState := E_Sercos_State.S7_FaultReactionActive;
	RETURN;
END_IF

IF NOT stControl.b15_Enable THEN 
	_eState := E_Sercos_State.S3_ReadyToSwitchOn;
	RETURN;
END_IF

IF NOT stControl.b14_Start THEN
	_eState := E_Sercos_State.S6_QuickStop;
	RETURN;
END_IF

IF NOT stControl.b13_Halt THEN
	_eState := E_Sercos_State.S5a_DriveInOperation;
	RETURN;
END_IF
END_METHOD

METHOD PRIVATE S6_QuickStop : BOOL
VAR_INPUT
END_VAR
stStatus.b15_ReadyToOperate 		:= TRUE;
stStatus.b14_ReadyToOperate 		:= TRUE;
stStatus.b13_Error 					:= FALSE;
stStatus.b7_QuickStop 				:= TRUE;
stStatus.b4_Halt 					:= TRUE;
stStatus.b3_CommandProcessing 		:= FALSE;

IF NOT bPower THEN
	_eState := E_Sercos_State.S2_SwitchOnDisabled;
	RETURN;
END_IF

IF _bError THEN
	_eState := E_Sercos_State.S7_FaultReactionActive;
	RETURN;
END_IF

IF NOT stControl.b15_Enable THEN 
	_eState := E_Sercos_State.S3_ReadyToSwitchOn;
	RETURN;
END_IF

IF stControl.b13_Halt AND stControl.b14_Start THEN
	_eState := E_Sercos_State.S5b_Halt;
	RETURN;
END_IF

IF NOT stControl.b13_Halt AND stControl.b14_Start THEN
	_eState := E_Sercos_State.S5a_DriveInOperation;
	RETURN;
END_IF
END_METHOD

METHOD PRIVATE S7_FaultReactionActive : BOOL
VAR_INPUT
END_VAR
stStatus.b15_ReadyToOperate 		:= TRUE;
stStatus.b14_ReadyToOperate 		:= TRUE;
stStatus.b13_Error 					:= TRUE;
stStatus.b7_QuickStop 				:= FALSE;
stStatus.b4_Halt 					:= FALSE;
stStatus.b3_CommandProcessing 		:= FALSE;

IF NOT bPower THEN
	_eState := E_Sercos_State.S2_SwitchOnDisabled;
	RETURN;
END_IF

_eState := E_Sercos_State.S8_Fault;
END_METHOD

METHOD PRIVATE S8_Fault : BOOL
VAR_INPUT
END_VAR
stStatus.b15_ReadyToOperate 		:= TRUE;
stStatus.b14_ReadyToOperate 		:= FALSE;
stStatus.b13_Error 					:= TRUE;
stStatus.b7_QuickStop 				:= FALSE;
stStatus.b4_Halt 					:= FALSE;
stStatus.b3_CommandProcessing 		:= FALSE;

IF _rTrig_Reset.Q THEN
	_eState := E_Sercos_State.S2_SwitchOnDisabled;
	_bError := FALSE;
	RETURN;	
END_IF
END_METHOD

END_FUNCTION_BLOCK

// ---- Tests/Drives/FB_Sercos_VC_Test.TcPOU
FUNCTION_BLOCK FB_Sercos_VC_Test EXTENDS TcUnit.FB_TestSuite

TestEnable();
TestEnableSTO();

TestGetProccesData('Get Process Data', FALSE);
TestGetProccesData('Get Process Data Swap', TRUE);
TestSetProccesData('Set Process Data', FALSE);
TestSetProccesData('Set Process Data Swap', TRUE);

TestCaseGetVelocity('Get Velocity 1', 80000, 2000, 80000, 2000);
TestCaseGetVelocity('Get Velocity 2', 40000, 2000, 80000, 1000);
TestCaseGetVelocity('Get Velocity 3', 0, 2000, 80000, 0);
TestCaseGetVelocity('Get Velocity 4', -40000, 2000, 80000, -1000);
TestCaseGetVelocity('Get Velocity 5', -80000, 2000, 80000, -2000);
TestCaseGetVelocity('Get Velocity 6', 80000, 500, 80000, 500);
TestCaseGetVelocity('Get Velocity 7', -80000, 500, 80000, -500);

METHOD PRIVATE EnableSequence : REFERENCE TO FB_Test
VAR_INPUT
	fbDrive : REFERENCE TO FB_Sercos_VC;
END_VAR
fbDrive.stControl.nControlWord.b13_Halt := FALSE;
fbDrive.stControl.nControlWord.b14_Start := TRUE;
fbDrive.stControl.nControlWord.b15_Enable := TRUE;

fbDrive();
fbDrive();
fbDrive();
fbDrive();
END_METHOD

METHOD TestCaseGetVelocity
VAR_INPUT
	sName : T_MaxString;	
	nVelocityCommand 			: DINT;
	fReferenceVelocity			: REAL;
	nNormalizationFactor 		: REAL;	
	fExpected 					: LREAL;
END_VAR

VAR	
	fbDrive		: FB_Sercos_VC;
	fResult 	: LREAL;
END_VAR
TEST(sName);
	

fResult := fbDrive.GetTargetVelocity(nVelocityCommand, fReferenceVelocity, nNormalizationFactor);
AssertEquals(Expected := fExpected,
             Actual := fResult,
             Message := 'Result value is not correct');	
	 
TEST_FINISHED();
END_METHOD

METHOD TestEnable : BOOL
VAR
	fbDrive 			: FB_Sercos_VC;	
	nActualState		: INT;
	nExpectedState		: INT;
END_VAR
TEST('Enable STO FALSE');
fbDrive.bSTO := FALSE;

EnableSequence(fbDrive);

nExpectedState := E_Sercos_State.S2_SwitchOnDisabled;
nActualState := fbDrive.eState;

AssertEquals(Expected := nExpectedState,
             Actual := nActualState,
             Message := 'State is not correct');	 
TEST_FINISHED();
END_METHOD

METHOD TestEnableSTO : BOOL
VAR
	fbDrive 			: FB_Sercos_VC;	
	nActualState		: INT;
	nExpectedState		: INT;
END_VAR
TEST('Enable STO TRUE');
fbDrive.bSTO := TRUE;
EnableSequence(fbDrive);

nExpectedState := E_Sercos_State.S5a_DriveInOperation;
nActualState := fbDrive.eState;

AssertEquals(Expected := nExpectedState,
             Actual := nActualState,
             Message := 'State is not correct');	 
TEST_FINISHED();
END_METHOD

METHOD TestGetProccesData : REFERENCE TO FB_Test
VAR_INPUT
	sName 					: T_MaxString;
	bSwap					: BOOL;
END_VAR

VAR
	fbDrive 				: FB_Sercos_VC;
	
	aControlData			: ARRAY [0..12] OF BYTE;
	aStatusData				: ARRAY [0..12] OF BYTE;
	
	nControlWordExpected	: WORD; 
	nControlWordActual		: WORD; 
	nTargetExpected			: DINT; 
	nTargetActual			: DINT;	
END_VAR
TEST(sName);

fbDrive.stConfig.bSwapProcessData := bSwap;
fbDrive.pControl := ADR(aControlData);
fbDrive.pStatus := ADR(aStatusData);

nControlWordExpected := 156;
nTargetExpected := 15674;
F_Memcpy(ADR(aControlData), ADR(nControlWordExpected), SIZEOF(nControlWordExpected), bSwap);
F_Memcpy(ADR(aControlData) + 2, ADR(nTargetExpected), SIZEOF(nTargetExpected), bSwap);

fbDrive.GetControlData();

F_Memcpy(ADR(nControlWordActual), ADR(fbDrive.stControl.nControlWord), SIZEOF(fbDrive.stControl.nControlWord), FALSE);
nTargetActual := fbDrive.stControl.nVelocityCommand;

AssertEquals_WORD(Expected := nControlWordExpected,
             Actual := nControlWordActual,
             Message := 'nControlWord is not correct');	

AssertEquals_DINT(Expected := nTargetExpected,
             Actual := nTargetActual,
             Message := '.nVelocityCommand is not correct');	

TEST_FINISHED();
END_METHOD

METHOD TestSetProccesData : REFERENCE TO FB_Test
VAR_INPUT
	sName 					: T_MaxString;
	bSwap					: BOOL;
END_VAR

VAR
	fbDrive 				: FB_Sercos_VC;
	
	aControlData			: ARRAY [0..12] OF BYTE;
	aStatusData				: ARRAY [0..12] OF BYTE;
	
	nStatusWordExpected		: WORD; 
	nStatusWordActual		: WORD; 
	nActualExpected			: DINT; 
	nActualActual			: DINT;
END_VAR
TEST(sName);

fbDrive.stConfig.bSwapProcessData := bSwap;
fbDrive.pControl := ADR(aControlData);
fbDrive.pStatus := ADR(aStatusData);

nStatusWordExpected := 156;
nActualExpected := 15674;

F_Memcpy(ADR(fbDrive.stStatus), ADR(nStatusWordExpected), SIZEOF(nStatusWordExpected), FALSE);
F_Memcpy(ADR(fbDrive.stStatus) + 2, ADR(nActualExpected), SIZEOF(nActualExpected), FALSE);

fbDrive.SetStatusData();

F_Memcpy(ADR(nStatusWordActual), ADR(aStatusData), SIZEOF(nStatusWordActual), bSwap);
F_Memcpy(ADR(nActualActual), ADR(aStatusData) + 2, SIZEOF(nActualActual), bSwap);


AssertEquals_WORD(Expected := nStatusWordExpected,
             Actual := nStatusWordActual,
             Message := 'nStatusWord is not correct');	

AssertEquals_DINT(Expected := nActualExpected,
             Actual := nActualActual,
             Message := '.nActualPosition is not correct');	

TEST_FINISHED();
END_METHOD

END_FUNCTION_BLOCK

// ---- Devices/Drives/Sercos/FB_Sercos_VC.TcPOU
(*
	Sercos Velocity Control
	MDT: S-0-0134 Master control word
	MDT: S-0-0036 Velocity command value
	AT: S-0-0135 Drive Status word
	AT: S-0-0051 Position feedback 1 value
*)

{attribute 'reflection'} 
FUNCTION_BLOCK FB_Sercos_VC EXTENDS FB_LinkDataReal 
VAR_INPUT
	pControl			: PVOID; //Pocess data from fieldbus, 4 BYTES FROM FIELDBUS
	pStatus				: PVOID; //Pocess data to fieldbus, 4 BYTES FROM FIELDBUS		
	stControl	 		: ST_Sercos_VC_Control;
	stConfig			: ST_Sercos_VC_Config;
	bSTO 				: BOOL := TRUE;
END_VAR

VAR_OUTPUT
	stStatus 			: ST_Sercos_VC_Status;	
END_VAR

VAR		
	{attribute 'instance-path'} 
    {attribute 'noinit'} 
    _sPath 				: STRING;
	_fbStateMachine 	: FB_Sercos_FSM;
	_fbEncoder 			: FB_Encoder;	
	_fVelocity			: REAL;
END_VAR

SUPER^();
InitRun();

GetControlData();
Cycle();
SetStatusData();

METHOD PRIVATE Cycle
VAR
	fTargetVelocitySign : REAL;
	fTargetVelocityFactor : REAL;
	fTargetVelocity : REAL;	
END_VAR
_fbStateMachine.bPower := bSTO;

_fbStateMachine.stControl := stControl.nControlWord;
_fbStateMachine();
stStatus.nStatusWord := _fbStateMachine.stStatus;

IF (_fbStateMachine._eState = E_Sercos_State.S5a_DriveInOperation OR _fbStateMachine._eState = E_Sercos_State.S5b_Halt) THEN	
	_fbEncoder.fValue := _fVelocity := GetTargetVelocity(stControl.nVelocityCommand, stConfig.fReferenceVelocity, stConfig.fNormalizationFactor);	
	_fbEncoder();
END_IF

stStatus.nStatusWord.b8_Reserved := stControl.nControlWord.b8_Reserved;
stStatus.nStatusWord.b9_Reserved := stControl.nControlWord.b9_Reserved;
stStatus.nStatusWord.b10_OperationMode := stControl.nControlWord.b11_Reserved;

stStatus.nPositionFeedback := _fbEncoder.nResult;

//Set Link Data
IF stConfig.bIsLinkOutputVelocity THEN
	ControlData := LREAL_TO_REAL(_fVelocity);
ELSE
	ControlData := LREAL_TO_REAL(_fbEncoder.fResult);
END_IF
END_METHOD

PROPERTY eState : E_Sercos_State
GET
eState := _fbStateMachine.eState;
END_GET
END_PROPERTY

PROPERTY PUBLIC fbEncoder : REFERENCE TO FB_Encoder
GET
fbEncoder REF= _fbEncoder;
END_GET
END_PROPERTY

METHOD INTERNAL GetControlData
IF pControl <= 0 OR stConfig.bForceMode THEN RETURN; END_IF

(*Control Word*)
F_Memcpy(ADR(stControl), pControl, 2, stConfig.bSwapProcessData);
(*Velocity Command*)
F_Memcpy(ADR(stControl) + 2, pControl + 2, 4, stConfig.bSwapProcessData);
END_METHOD

METHOD INTERNAL GetTargetVelocity : REAL
VAR_INPUT
	nVelocityCommand 			: DINT;
	fReferenceVelocity			: REAL;
	nNormalizationFactor 		: REAL;
END_VAR

VAR
	fTargetVelocity 			: REAL;	
	fTargetVelocitySign 		: REAL;
	fTargetVelocityFactor 		: REAL;	
END_VAR
fTargetVelocity := DINT_TO_REAL(nVelocityCommand);
fTargetVelocityFactor := F_Norm(0, nNormalizationFactor, ABS(fTargetVelocity));
GetTargetVelocity := fReferenceVelocity * fTargetVelocityFactor * F_Sign(fTargetVelocity);
END_METHOD

METHOD PRIVATE InitRun
VAR_INST
	bInitRun : BOOL := TRUE;
END_VAR
IF NOT bInitRun THEN RETURN; END_IF
bInitRun := FALSE;

IF pControl = 0 OR pStatus = 0 THEN
	ADSLOGSTR(ADSLOG_MSGTYPE_WARN, '%s', CONCAT(_sPath, ' PLC IO is not assigned!'));	
END_IF

_fbEncoder.stConfig.bIsIntegrator := TRUE;
END_METHOD

METHOD PRIVATE Motion : REAL
VAR_INPUT
END_VAR
END_METHOD

METHOD INTERNAL SetStatusData
IF pStatus <= 0 THEN RETURN; END_IF

(*StatusWord*)
F_Memcpy(pStatus, ADR(stStatus), 2, stConfig.bSwapProcessData);
(*Position Feedback*)
F_Memcpy(pStatus + 2, ADR(stStatus) + 2, 4, stConfig.bSwapProcessData);
END_METHOD

END_FUNCTION_BLOCK

// ---- Devices/Drives/Mitsubishi/FB_Mitsubishi_MRJ4TM.TcPOU
(*
	
